// SIMATIC STEP 7 (V5.x) project 2800
// CPU: CPU 315-2 DP
// station: P_ADR_BUS
// station: Hardware
// station: SIMATIC 300(1)
// program: S7 Program(1)

SYMBOL_TABLE
"CLOCK_OP"	DB 5	DB 5	// COMMUNICATION CLOCK OP
"TransferValves"	DB 10	DB 10	// Data Transfer for Valves
"TransferMotor"	DB 11	DB 11	// Data Transfer for Motor
"TransferLevel"	DB 12	DB 12	// Data Transfer for Level
"TransferTemperature"	DB 14	DB 14	// Data Transfer for Temperatuer
"TransferPID"	DB 15	DB 15	// Data Transfer for PID
"TransferFlow"	DB 16	DB 16	// Data Transfer for Flow
"TransferWeight"	DB 18	DB 18	// Data Transfer for Weight
"TransferGenerell"	DB 30	DB 30	// Data Transfer Generell
"TransferRecipe"	DB 90	DB 90	// Data Transfer for Recipe
"TransferBatch"	DB 91	DB 91	// Data Transfer for Batch
"DataBatchControl"	DB 92	FB 90
"ALARMTIME"	DB 100	DB 100	// actual timers alarms
"ALARMBLOCK"	DB 110	DB 110	// alarm indication to OP
"ALARM_ACK_OP"	DB 115	DB 115	// alarm acknowledge from OP
"LAMPS_ACK"	DB 120	DB 120	// lamp acknowledge
"CLOCK_FB"	FB 5	FB 5	// SETTING CPU CLOCK
"preparation"	FB 10	FB 10	// starch preparation
"Devices"	FB 20	FB 20	// Devices
"ALARM_HANDLING"	FB 31	FB 31	// alarm handling
"ALARM"	FB 33	FB 33	// indication alarm
"Batch"	FB 90	FB 90	// Batch
"BatchControl"	FC 10	FC 10	// Batch Control
"RecipeControl"	FC 90	FC 90	// Recipe Control
"DosLine"	FC 91	FC 91	// Dosing Line
"AUTO_VALVE"	FC 100	FC 100	// automatic valve
"MOTOR"	FC 101	FC 101	// motor control
"level"	FC 107	FC 107	// level display
"temperature"	FC 109	FC 109	// temperature display
"AI_4-20"	FC 111	FC 111	// analog input 4-20mA
"weight"	FC 114	FC 114	// weighing unit
"ALARM_BLOCK"	FC 115	FC 115	// alarm function block
"M22_01_RUN"	I 4.0	BOOL	// screw conveyor sizing starch running
"M23_01_RUN"	I 4.1	BOOL	// dedusting station sizing starch running
"M24_01_RUN"	I 4.2	BOOL	// agitator cooker sizing starch running
"M25_01_RUN"	I 4.3	BOOL	// pump sizing starch running
"M26_01_RUN"	I 4.4	BOOL	// stby pump sizing starch running
"HS22_02_ZSC"	I 4.5	BOOL	// valve screw conveyor sizing starch closed
"HS22_02_ZSO"	I 4.6	BOOL	// valve screw conveyor sizing starch open
"HS24_06_ZSC"	I 4.7	BOOL	// water valve cooker sizing starch closed
"HS24_08_ZSC"	I 5.0	BOOL	// discharge valve cooker sizing starch closed
"XS28_02_K1"	I 5.1	BOOL	// release filling storage tank sizing starch
"Signal_0"	M 1.0	BOOL	// Signal 0
"Signal_1"	M 1.1	BOOL	// Signal 1
"1_second"	M 1.2	BOOL	// second pulse
"PB_LAMP_ACK"	M 1.3	BOOL	// Lamp acknowledge
"spike_ pulse_ 1H"	M 2.0	BOOL	// spike pulse 1 houre
"Release_Time"	M 2.1	BOOL	// release timetransfer
"Pulse_Time"	M 2.2	BOOL	// pulse timetransfer
"OP_COMM_OK"	M 9.0	BOOL	// Op Communication ok
"LB_OP_PULS"	M 9.1	BOOL
"fault_M_22_01"	M 12.0	BOOL	// fault motor M 22.01
"fault_M_23_01"	M 12.1	BOOL	// fault motor M 23.01
"fault_M_24_01"	M 12.2	BOOL	// fault motor M 24.01
"fault_M_25_01"	M 12.3	BOOL	// fault motor M 25.01
"fault_M_26_01"	M 12.4	BOOL	// fault motor M 26.01
"fault_HS_22_02"	M 14.0	BOOL	// fault valve HS 22.02
"fault_HS_22_06"	M 14.1	BOOL	// fault valve HS 22.06
"fault_HS_24_06"	M 14.2	BOOL	// fault valve HS 24.06
"fault_HS_24_07"	M 14.3	BOOL	// fault valve HS 24.07
"fault_HS_24_08"	M 14.4	BOOL	// fault valve HS 24.08
"fault_WQ_24_04"	M 16.0	BOOL	// fault weighing unit WQ 24.04
"fault_TC_24_05"	M 16.1	BOOL	// fault temperature TC 24.05
"fault_XS_28_02"	M 16.2	BOOL	// fault level XS 28.02
"fault_HH_WQ_24_04"	M 17.0	BOOL	// fault alarm high weighing unit WQ 24.04
"fault_HH_TC_24_05"	M 17.1	BOOL	// fault alarm high temperature TC 24.05
"fault_HH_XS_28_02"	M 17.2	BOOL	// fault alarm high level XS 28.02
"fault_LL_XS_28_02"	M 17.3	BOOL	// fault alarm low level XS 28.02
"HH_WQ_24_04"	M 60.0	BOOL	// Alarm HH WQ 24.04
"HH_TC_24_05"	M 60.1	BOOL	// Alarm HH TC 24.05
"HH_XS_28_02"	M 60.2	BOOL	// Alarm HH XS 28.02
"H_WQ_24_05"	M 61.0	BOOL	// Alarm H WQ 24.05
"H_TC_24_05"	M 61.1	BOOL	// Alarm H TC 24.05
"H_XS_28_02"	M 61.2	BOOL	// Alarm H XS 28.02
"L_WQ_24_06"	M 62.0	BOOL	// Alarm L WQ 24.06
"L_TC_24_05"	M 62.1	BOOL	// Alarm L TC 24.05
"L_XS_28_02"	M 62.2	BOOL	// Alarm L XS 28.02
"LL_WQ_24_07"	M 63.0	BOOL	// Alarm LL WQ 24.07
"LL_TC_24_05"	M 63.1	BOOL	// Alarm LL TC 24.05
"LL_XS_28_02"	M 63.2	BOOL	// Alarm LL XS 28.02
"check_M_22_01"	M 70.0	BOOL	// check motor M 22.01
"check_M_23_01"	M 70.1	BOOL	// check motor M 23.01
"check_M_24_01"	M 70.2	BOOL	// check motor M 24.01
"check_M_25_01"	M 70.3	BOOL	// check motor M 25.01
"check_M_26_01"	M 70.4	BOOL	// check motor M 26.01
"check_HS_22_02"	M 72.0	BOOL	// check valve HS 22.02
"check_HS_22_06"	M 72.1	BOOL	// check valve HS 22.06
"check_HS_24_06"	M 72.2	BOOL	// check valve HS 24.06
"check_HS_24_07"	M 72.3	BOOL	// check valve HS 24.07
"check_HS_24_08"	M 72.4	BOOL	// check valve HS 24.08
"check_WQ_24_04"	M 74.0	BOOL	// check weight WQ 24.04
"check_TC_24_05"	M 74.1	BOOL	// check temperature TC 24.05
"check_XS_28_02"	M 74.2	BOOL	// check level XS 28.02
"fault_ack_M_22_01"	M 90.0	BOOL	// fault acknowledge motor M 22.01
"fault_ack_M_23_01"	M 90.1	BOOL	// fault acknowledge motor M 23.01
"fault_ack_M_24_01"	M 90.2	BOOL	// fault acknowledge motor M 24.01
"fault_ack_M_25_01"	M 90.3	BOOL	// fault acknowledge motor M 25.01
"fault_ack_M_26_01"	M 90.4	BOOL	// fault acknowledge motor M 26.01
"fault_ack_HS_22_02"	M 92.0	BOOL	// fault acknowledge valve HS 22.02
"fault_ack_HS_22_06"	M 92.1	BOOL	// fault acknowledge valve HS 22.06
"fault_ack_HS_24_06"	M 92.2	BOOL	// fault acknowledge valve HS 24.06
"fault_ack_HS_24_07"	M 92.3	BOOL	// fault acknowledge valve HS 24.07
"fault_ack_HS_24_08"	M 92.4	BOOL	// fault acknowledge valve HS 24.08
"fault_ack_WQ_24_04"	M 94.0	BOOL	// fault acknowledge weight WQ 24.04
"fault_ack_TC_24_05"	M 94.1	BOOL	// fault acknowledge temperature TC 24.05
"fault_ack_XS_28_02"	M 94.2	BOOL	// fault acknowledge level XS 28.02
"fault_ack_HH_WQ_24_04"	M 95.0	BOOL	// fault acknowledge alarm high weighing unit WQ 24.04
"fault_ack_HH_TC_24_05"	M 95.1	BOOL	// fault acknowledge alarm high temperature TC 24.05
"fault_ack_HH_XS_28_02"	M 95.2	BOOL	// fault acknowledge alarm high level XS 28.02
"fault_ack_LL_XS_28_02"	M 95.3	BOOL	// fault acknowledge alarm low level XS 28.02
"auto_on_M_22_01"	M 100.0	BOOL	// auto on motor M 22.01
"auto_on_M_23_01"	M 100.1	BOOL	// auto on motor M 23.01
"auto_on_M_24_01"	M 100.2	BOOL	// auto on motor M 24.01
"auto_on_M_25_01"	M 100.3	BOOL	// auto on motor M 25.01
"auto_on_M_26_01"	M 100.4	BOOL	// auto on motor M 26.01
"auto_on_HS_22_02"	M 102.0	BOOL	// auto on valve HS 22.02
"auto_on_HS_22_06"	M 102.1	BOOL	// auto on valve HS 22.06
"auto_on_HS_24_06"	M 102.2	BOOL	// auto on valve HS 24.06
"auto_on_HS_24_07"	M 102.3	BOOL	// auto on valve HS 24.07
"auto_on_HS_24_08"	M 102.4	BOOL	// auto on valve HS 24.08
"SteamOnEnzym"	M 102.5	BOOL	// Cond. Steam on if Enzymatic Starch selected
"AlarmOnEnzym"	M 102.6	BOOL	// Alarm On Enzym Dosing
"SteamOnHold"	M 102.7	BOOL	// Cond. Steam on at end Temperaturcontrol
"LockSelModified"	M 110.0	BOOL	// Lock Selection Button if Batch is running
"Cond_Dos_Starch"	M 120.0	BOOL	// Condition Dosing Starch
"Save_Dil_On_Starch"	M 120.1	BOOL	// Save Dilution was on starch
"Agitator_Stop_Starch"	M 120.2	BOOL	// Agitator stop starch
"Save_Dis_On_Starch"	M 120.3	BOOL	// Save discharge was on starch
"IMP_START_STARCH"	M 160.0	BOOL	// Impuls Start Batch Starch
"Hold_Mixing_Time_Starch"	M 160.1	BOOL	// Hold Mixing Time Starch
"Discharged1_Starch"	M 161.0	BOOL	// Discharged 1 starch
"Discharged2_Starch"	M 161.1	BOOL	// Discharged 2 starch
"Batch_Starch_Running"	M 180.0	BOOL	// Batch Starch Running
"Batch_Starch_Started"	M 180.1	BOOL	// Batch Starch Started
"Dos_On_Water_Starch"	M 185.0	BOOL	// Dosing on water starch
"Cmd_Agitator_On_Starch"	M 185.1	BOOL	// Command Agitator on starch
"Dos_On_Powder_Starch"	M 185.2	BOOL	// Dosing on powder starch
"Dos_On_Steam_Starch"	M 185.3	BOOL	// Dosing on steam starch
"Dos_On_Dil_Water_Starch"	M 185.4	BOOL	// Dosing on dilution water starch
"Cmd_Discharge1_On_Starch"	M 185.5	BOOL	// Command discharge 1 on starch
"Active_Discharge1_Starch"	M 185.6	BOOL	// Active Discharge 1 Starch
"Dos_On_Flushwater_Starch"	M 185.7	BOOL	// Dosing on flushwater starch
"Cmd_Discharge2_On_Starch"	M 186.0	BOOL	// Command discharge 2 on starch
"Active_Discharge2_Starch"	M 186.1	BOOL	// Active Discharge 2 Starch
"Active_Dil_Water_Starch"	M 186.2	BOOL	// Dosing active dilution water starch
"Cmd_Enzym_On_Starch"	M 186.3	BOOL	// Dosing Enzym Request
"Enzyme_Done_Starch"	M 186.4	BOOL	// Enzym finished
"Dos_On_EnzSteam_Starch"	M 186.5	BOOL	// Dosing on Steam for Enzymatic Starch
"Active_Hold_Temp_Starch"	M 186.6	BOOL	// Holding Temperature active Enzymatic Starch
"Active_Temp_Starch"	M 186.7	BOOL	// Temperature Hold at end of Starch
"WQ_24_04_Value"	MD 30	REAL	// value WQ 24.04
"TC_24_05_Value"	MD 34	REAL	// value TC 24.05
"XS_28_02_Value"	MD 38	REAL	// value percent XS 28.02
"Cycle_Time"	MW 252	INT	// Cycle Time
"WQ24_04_IN"	PIW 256	WORD	// weight cooker sizing starch
"XS28_02_LI"	PIW 258	WORD	// level storage tank cooked sizing starch
"TC24_05_IN"	PIW 260	WORD	// temperature cooker sizing starch
"M22_01_ON"	Q 8.0	BOOL	// screw conveyor sizing starch on
"M23_01_ON"	Q 8.1	BOOL	// dedusting station sizing starch on
"M23_01_ST"	Q 8.2	BOOL	// dedusting station sizing starch on
"M24_01_ON"	Q 8.3	BOOL	// agitator cooker sizing starch on
"M25_01_ON"	Q 8.4	BOOL	// pump sizing starch on
"M26_01_ON"	Q 8.5	BOOL	// stby pump sizing starch on
"HS22_02_ON"	Q 8.6	BOOL	// valve screw conveyor sizing starch on
"HS22_06_ON"	Q 8.7	BOOL	// air valve screw conveyor sizing starch on
"HS24_06_ON"	Q 9.0	BOOL	// water valve cooker sizing starch on
"HS24_07_ON"	Q 9.1	BOOL	// steam valve cooker sizing starch on
"HS24_08_ON"	Q 9.2	BOOL	// discharge valve cooker sizing starch on
"XA28_01_ON"	Q 9.3	BOOL	// alarm preparation on
"XS28_02_K2"	Q 9.4	BOOL	// filling is on storage tank sizing starch
"XS28_02_K3"	Q 9.5	BOOL	// fault filling storage tank sizing starch
"SET_CLK"	SFC 0	SFC 0	// Set System Clock
"Valve UDT"	UDT 1	UDT 1	// Data Valve
"Valve Popup UDT"	UDT 2	UDT 2	// Data Valve Popup
"Motor UDT"	UDT 3	UDT 3	// Data Motor
"Motor Popup UDT"	UDT 4	UDT 4	// Data Motor Popup
"Level UDT"	UDT 5	UDT 5	// Data Level
"Level Popup UDT"	UDT 6	UDT 6	// Data Level Popup
"Pressure UDT"	UDT 7	UDT 7	// Data Pressure
"Pressure Popup UDT"	UDT 8	UDT 8	// Data Pressure Popup
"Temperature UDT"	UDT 9	UDT 9	// Data Temperature
"Temperature Popup UDT"	UDT 10	UDT 10	// Data Temperature Popup
"Controler UDT"	UDT 11	UDT 11	// Data Controler
"Controler Popup UDT"	UDT 12	UDT 12	// Data Controler Popup
"Flow UDT"	UDT 13	UDT 13	// Data Flow
"Flow Popup UDT"	UDT 14	UDT 14	// Data Flow Popup
"Viskosity UDT"	UDT 15	UDT 15	// Viskosity Data
"Viskosity Popup UDT"	UDT 16	UDT 16	// Data Viskosity Popup
"Weight UDT"	UDT 17	UDT 17	// Weight Data
"Weight Popup UDT"	UDT 18	UDT 18	// Data Weight Popup
"Recipe UDT"	UDT 90	UDT 90	// Data Recipe
"DosLine UDT"	UDT 91	UDT 91	// Dosing Line UDT
END_SYMBOL_TABLE

FUNCTION_BLOCK "CLOCK_FB"	// FB 5
AUTHOR : gaw-be
FAMILY : GAW
NAME : DATETIME
VERSION : 0.1
BEGIN
// (block stored without names or comments; labels and parameter names are numbered)
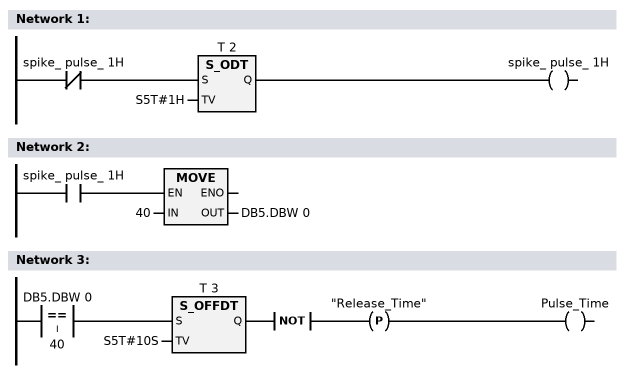
NETWORK
TITLE =
      AN    "spike_ pulse_ 1H";
      L     S5T#1H;
      SD    T 2;
      NOP   0;
      NOP   0;
      NOP   0;
      A     T 2;
      =     "spike_ pulse_ 1H";
NETWORK
TITLE =
      A     "spike_ pulse_ 1H";
      JNB   M001;
      L     40;
      T     DB5.DBW 0;
M001: NOP   0;
NETWORK
TITLE =
      A(;
      A(;
      L     DB5.DBW 0;
      L     40;
      ==I;
      );
      L     S5T#10S;
      SF    T 3;
      NOP   0;
      NOP   0;
      NOP   0;
      A     T 3;
      );
      NOT;
      FP    "Release_Time";
      =     "Pulse_Time";
NETWORK
TITLE =
      A     "Pulse_Time";
      JNB   M002;
      BLD   7;
      L     5;
      T     LW 102;
      L     P#DBX 8.0;
      T     LD 104;
      UC    "SET_CLK";
      {     P#L 102.0, P#L 100.0 };
      BLD   8;
M002: NOP   0;
END_FUNCTION_BLOCK

FUNCTION_BLOCK "preparation"	// FB 10
VERSION : 0.1
BEGIN
// (block stored without names or comments; labels and parameter names are numbered)
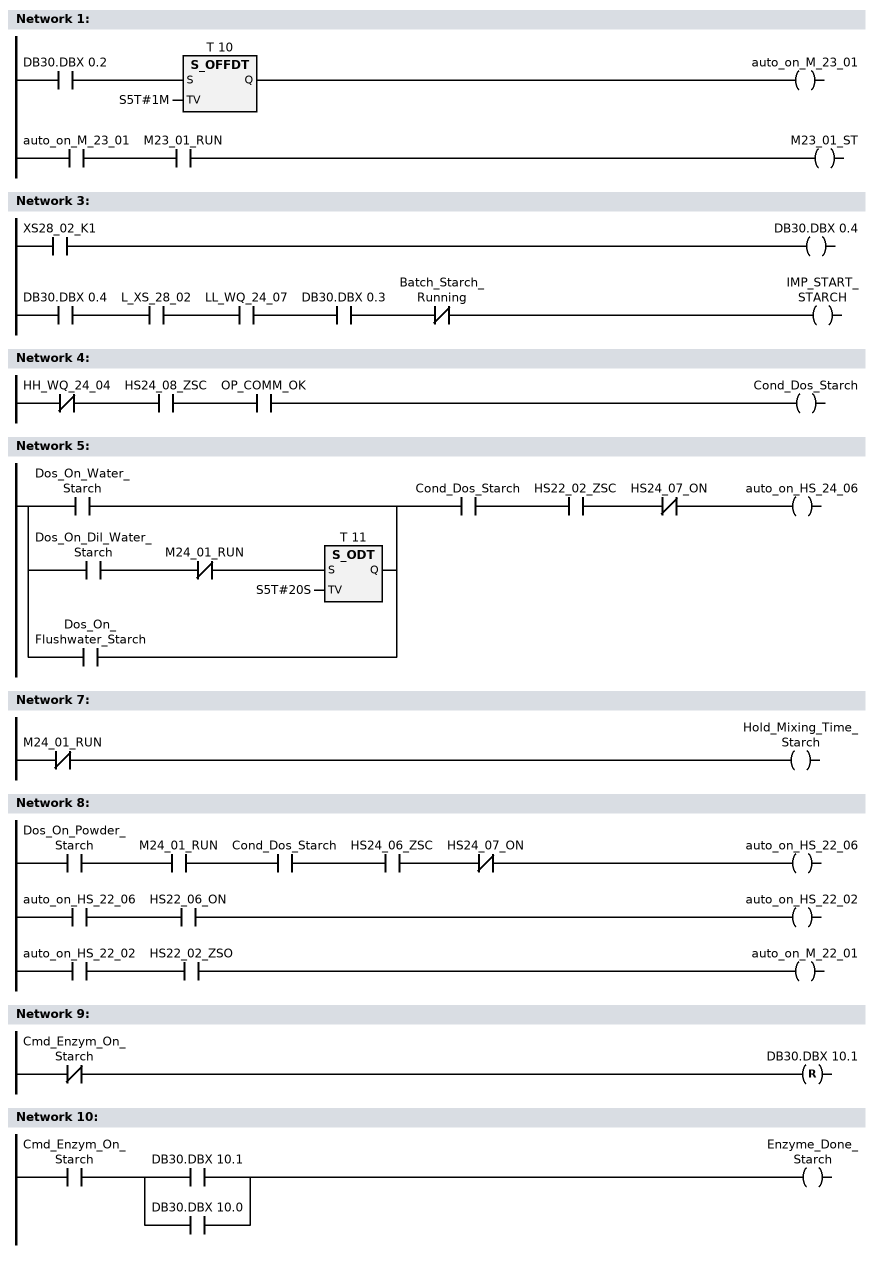
NETWORK
TITLE =
      A(;
      A     DB30.DBX 0.2;
      L     S5T#1M;
      SF    T 10;
      NOP   0;
      NOP   0;
      NOP   0;
      A     T 10;
      );
      =     "auto_on_M_23_01";
      A     "auto_on_M_23_01";
      A     "M23_01_RUN";
      =     "M23_01_ST";
NETWORK
TITLE =
      AN    "Batch_Starch_Running";
      A     DB30.DBX 10.0;
      S     "LockSelModified";
      AN    "Batch_Starch_Running";
      AN    DB30.DBX 10.0;
      R     "LockSelModified";
      A     "LockSelModified";
      =     L 8.0;
      A     L 8.0;
      A     "Batch_Starch_Running";
      S     DB30.DBX 10.0;
      AN    L 8.0;
      A     "Batch_Starch_Running";
      R     DB30.DBX 10.0;
NETWORK
TITLE =
      A     "XS28_02_K1";
      =     DB30.DBX 0.4;
      A     DB30.DBX 0.4;
      A     "L_XS_28_02";
      A     "LL_WQ_24_07";
      A     DB30.DBX 0.3;
      AN    "Batch_Starch_Running";
      =     "IMP_START_STARCH";
NETWORK
TITLE =
      AN    "HH_WQ_24_04";
      A     "HS24_08_ZSC";
      A     "OP_COMM_OK";
      =     "Cond_Dos_Starch";
NETWORK
TITLE =
      A(;
      O     "Dos_On_Water_Starch";
      O(;
      A     "Dos_On_Dil_Water_Starch";
      AN    "M24_01_RUN";
      L     S5T#20S;
      SD    T 11;
      NOP   0;
      NOP   0;
      NOP   0;
      A     T 11;
      );
      O     "Dos_On_Flushwater_Starch";
      );
      A     "Cond_Dos_Starch";
      A     "HS22_02_ZSC";
      AN    "HS24_07_ON";
      =     "auto_on_HS_24_06";
NETWORK
TITLE =
      AN    "LL_WQ_24_07";
      A     "Cmd_Agitator_On_Starch";
      A(;
      A(;
      A     "Dos_On_Dil_Water_Starch";
      S     "Save_Dil_On_Starch";
      AN    "Active_Dil_Water_Starch";
      R     "Save_Dil_On_Starch";
      A     "Save_Dil_On_Starch";
      );
      NOT;
      );
      A(;
      A(;
      A     "Cmd_Discharge1_On_Starch";
      A     "L_WQ_24_06";
      S     "Agitator_Stop_Starch";
      AN    "Batch_Starch_Running";
      R     "Agitator_Stop_Starch";
      A     "Agitator_Stop_Starch";
      );
      NOT;
      );
      =     "auto_on_M_24_01";
NETWORK
TITLE =
      AN    "M24_01_RUN";
      =     "Hold_Mixing_Time_Starch";
NETWORK
TITLE =
      A     "Dos_On_Powder_Starch";
      A     "M24_01_RUN";
      A     "Cond_Dos_Starch";
      A     "HS24_06_ZSC";
      AN    "HS24_07_ON";
      =     "auto_on_HS_22_06";
      A     "auto_on_HS_22_06";
      A     "HS22_06_ON";
      =     "auto_on_HS_22_02";
      A     "auto_on_HS_22_02";
      A     "HS22_02_ZSO";
      =     "auto_on_M_22_01";
NETWORK
TITLE =
      AN    "Cmd_Enzym_On_Starch";
      R     DB30.DBX 10.1;
NETWORK
TITLE =
      A     "Cmd_Enzym_On_Starch";
      A(;
      O     DB30.DBX 10.1;
      O     DB30.DBX 10.0;
      );
      =     "Enzyme_Done_Starch";
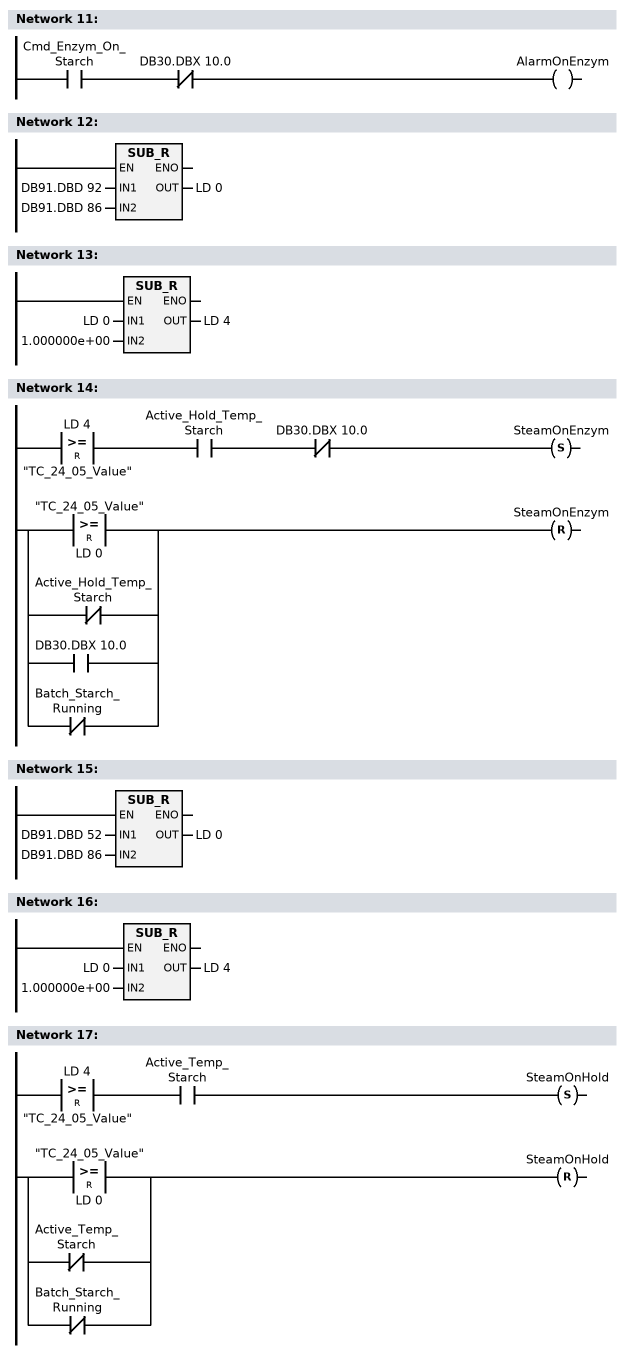
NETWORK
TITLE =
      A     "Cmd_Enzym_On_Starch";
      AN    DB30.DBX 10.0;
      =     "AlarmOnEnzym";
NETWORK
TITLE =
      L     DB91.DBD 92;
      L     DB91.DBD 86;
      -R;
      T     LD 0;
      NOP   0;
NETWORK
TITLE =
      L     LD 0;
      L     1.000000e+00;
      -R;
      T     LD 4;
      NOP   0;
NETWORK
TITLE =
      A(;
      L     LD 4;
      L     "TC_24_05_Value";
      >=R;
      );
      A     "Active_Hold_Temp_Starch";
      AN    DB30.DBX 10.0;
      S     "SteamOnEnzym";
      A(;
      O(;
      L     "TC_24_05_Value";
      L     LD 0;
      >=R;
      );
      ON    "Active_Hold_Temp_Starch";
      O     DB30.DBX 10.0;
      ON    "Batch_Starch_Running";
      );
      R     "SteamOnEnzym";
      NOP   0;
NETWORK
TITLE =
      L     DB91.DBD 52;
      L     DB91.DBD 86;
      -R;
      T     LD 0;
      NOP   0;
NETWORK
TITLE =
      L     LD 0;
      L     1.000000e+00;
      -R;
      T     LD 4;
      NOP   0;
NETWORK
TITLE =
      A(;
      L     LD 4;
      L     "TC_24_05_Value";
      >=R;
      );
      A     "Active_Temp_Starch";
      S     "SteamOnHold";
      A(;
      O(;
      L     "TC_24_05_Value";
      L     LD 0;
      >=R;
      );
      ON    "Active_Temp_Starch";
      ON    "Batch_Starch_Running";
      );
      R     "SteamOnHold";
      NOP   0;
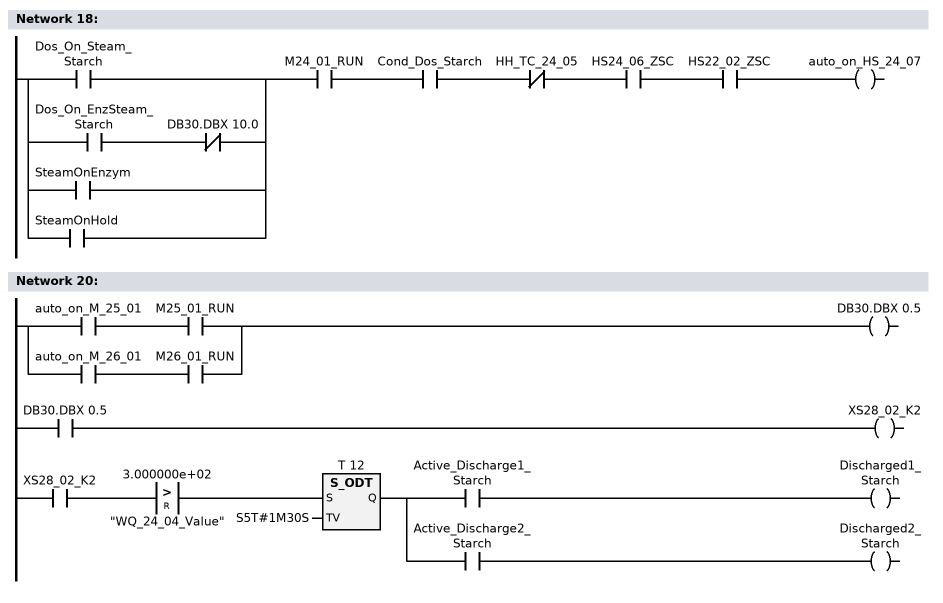
NETWORK
TITLE =
      A(;
      O     "Dos_On_Steam_Starch";
      O;
      A     "Dos_On_EnzSteam_Starch";
      AN    DB30.DBX 10.0;
      O     "SteamOnEnzym";
      O     "SteamOnHold";
      );
      A     "M24_01_RUN";
      A     "Cond_Dos_Starch";
      AN    "HH_TC_24_05";
      A     "HS24_06_ZSC";
      A     "HS22_02_ZSC";
      =     "auto_on_HS_24_07";
NETWORK
TITLE =
      A(;
      A(;
      A     "XS28_02_K1";
      A     "L_XS_28_02";
      O(;
      A     "auto_on_HS_24_08";
      A     "Active_Discharge1_Starch";
      S     "Save_Dis_On_Starch";
      AN    "Active_Discharge1_Starch";
      R     "Save_Dis_On_Starch";
      A     "Save_Dis_On_Starch";
      );
      );
      A     "Cmd_Discharge1_On_Starch";
      A     "Active_Discharge1_Starch";
      O;
      A     "Cmd_Discharge2_On_Starch";
      A     "Active_Discharge2_Starch";
      );
      AN    "HH_XS_28_02";
      =     "auto_on_HS_24_08";
      A     "auto_on_HS_24_08";
      AN    "HS24_08_ZSC";
      =     L 8.0;
      A     L 8.0;
      AN    DB30.DBX 0.0;
      =     "auto_on_M_25_01";
      A     L 8.0;
      A     DB30.DBX 0.0;
      =     "auto_on_M_26_01";
NETWORK
TITLE =
      A(;
      A     "auto_on_M_25_01";
      A     "M25_01_RUN";
      O;
      A     "auto_on_M_26_01";
      A     "M26_01_RUN";
      );
      =     DB30.DBX 0.5;
      A     DB30.DBX 0.5;
      =     "XS28_02_K2";
      A     "XS28_02_K2";
      A(;
      L     3.000000e+02;
      L     "WQ_24_04_Value";
      >R;
      );
      L     S5T#1M30S;
      SD    T 12;
      NOP   0;
      NOP   0;
      NOP   0;
      A     T 12;
      =     L 8.0;
      A     L 8.0;
      A     "Active_Discharge1_Starch";
      =     "Discharged1_Starch";
      A     L 8.0;
      A     "Active_Discharge2_Starch";
      =     "Discharged2_Starch";
END_FUNCTION_BLOCK

FUNCTION_BLOCK "Devices"	// FB 20
VERSION : 0.1
BEGIN
// (block stored without names or comments; labels and parameter names are numbered)
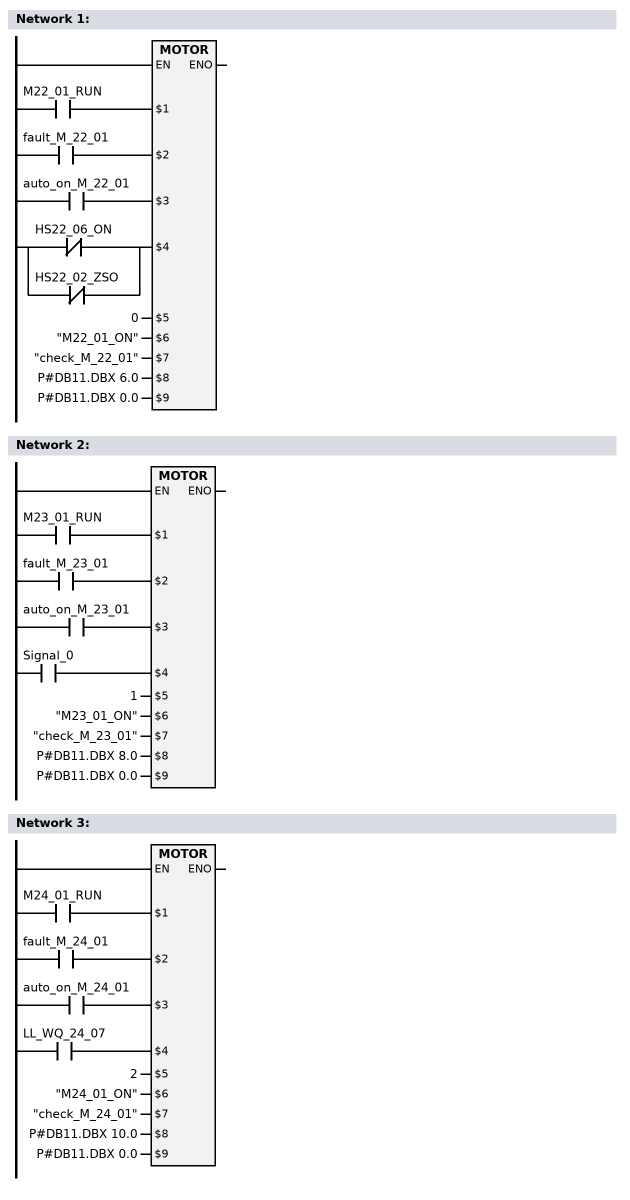
NETWORK
TITLE =
      A     "M22_01_RUN";
      =     L 18.0;
      BLD   103;
      A     "fault_M_22_01";
      =     L 18.1;
      BLD   103;
      A     "auto_on_M_22_01";
      =     L 18.2;
      BLD   103;
      A(;
      ON    "HS22_06_ON";
      ON    "HS22_02_ZSO";
      );
      =     L 18.3;
      BLD   103;
      CALL  "MOTOR" (
           $1                       := L 18.0,
           $2                       := L 18.1,
           $3                       := L 18.2,
           $4                       := L 18.3,
           $5                       := 0,
           $6                       := "M22_01_ON",
           $7                       := "check_M_22_01",
           $8                       := P#DB11.DBX 6.0,
           $9                       := P#DB11.DBX 0.0);
      NOP   0;
NETWORK
TITLE =
      A     "M23_01_RUN";
      =     L 18.0;
      BLD   103;
      A     "fault_M_23_01";
      =     L 18.1;
      BLD   103;
      A     "auto_on_M_23_01";
      =     L 18.2;
      BLD   103;
      A     "Signal_0";
      =     L 18.3;
      BLD   103;
      CALL  "MOTOR" (
           $1                       := L 18.0,
           $2                       := L 18.1,
           $3                       := L 18.2,
           $4                       := L 18.3,
           $5                       := 1,
           $6                       := "M23_01_ON",
           $7                       := "check_M_23_01",
           $8                       := P#DB11.DBX 8.0,
           $9                       := P#DB11.DBX 0.0);
      NOP   0;
NETWORK
TITLE =
      A     "M24_01_RUN";
      =     L 18.0;
      BLD   103;
      A     "fault_M_24_01";
      =     L 18.1;
      BLD   103;
      A     "auto_on_M_24_01";
      =     L 18.2;
      BLD   103;
      A     "LL_WQ_24_07";
      =     L 18.3;
      BLD   103;
      CALL  "MOTOR" (
           $1                       := L 18.0,
           $2                       := L 18.1,
           $3                       := L 18.2,
           $4                       := L 18.3,
           $5                       := 2,
           $6                       := "M24_01_ON",
           $7                       := "check_M_24_01",
           $8                       := P#DB11.DBX 10.0,
           $9                       := P#DB11.DBX 0.0);
      NOP   0;
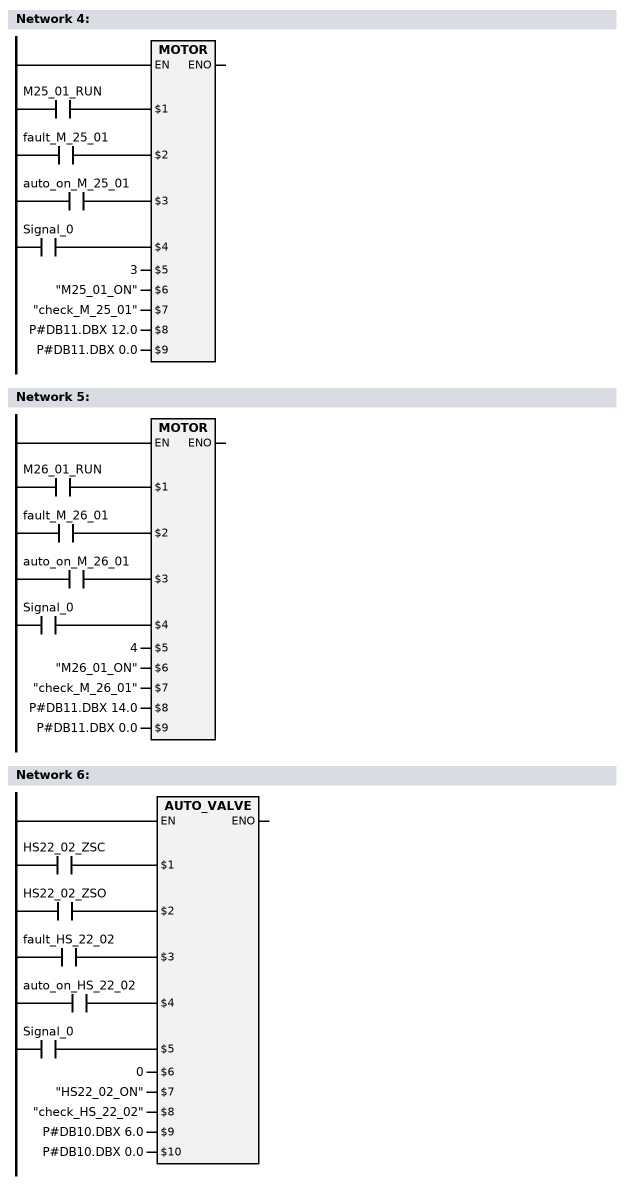
NETWORK
TITLE =
      A     "M25_01_RUN";
      =     L 18.0;
      BLD   103;
      A     "fault_M_25_01";
      =     L 18.1;
      BLD   103;
      A     "auto_on_M_25_01";
      =     L 18.2;
      BLD   103;
      A     "Signal_0";
      =     L 18.3;
      BLD   103;
      CALL  "MOTOR" (
           $1                       := L 18.0,
           $2                       := L 18.1,
           $3                       := L 18.2,
           $4                       := L 18.3,
           $5                       := 3,
           $6                       := "M25_01_ON",
           $7                       := "check_M_25_01",
           $8                       := P#DB11.DBX 12.0,
           $9                       := P#DB11.DBX 0.0);
      NOP   0;
NETWORK
TITLE =
      A     "M26_01_RUN";
      =     L 18.0;
      BLD   103;
      A     "fault_M_26_01";
      =     L 18.1;
      BLD   103;
      A     "auto_on_M_26_01";
      =     L 18.2;
      BLD   103;
      A     "Signal_0";
      =     L 18.3;
      BLD   103;
      CALL  "MOTOR" (
           $1                       := L 18.0,
           $2                       := L 18.1,
           $3                       := L 18.2,
           $4                       := L 18.3,
           $5                       := 4,
           $6                       := "M26_01_ON",
           $7                       := "check_M_26_01",
           $8                       := P#DB11.DBX 14.0,
           $9                       := P#DB11.DBX 0.0);
      NOP   0;
NETWORK
TITLE =
      A     "HS22_02_ZSC";
      =     L 18.0;
      BLD   103;
      A     "HS22_02_ZSO";
      =     L 18.1;
      BLD   103;
      A     "fault_HS_22_02";
      =     L 18.2;
      BLD   103;
      A     "auto_on_HS_22_02";
      =     L 18.3;
      BLD   103;
      A     "Signal_0";
      =     L 18.4;
      BLD   103;
      CALL  "AUTO_VALVE" (
           $1                       := L 18.0,
           $2                       := L 18.1,
           $3                       := L 18.2,
           $4                       := L 18.3,
           $5                       := L 18.4,
           $6                       := 0,
           $7                       := "HS22_02_ON",
           $8                       := "check_HS_22_02",
           $9                       := P#DB10.DBX 6.0,
           $10                      := P#DB10.DBX 0.0);
      NOP   0;
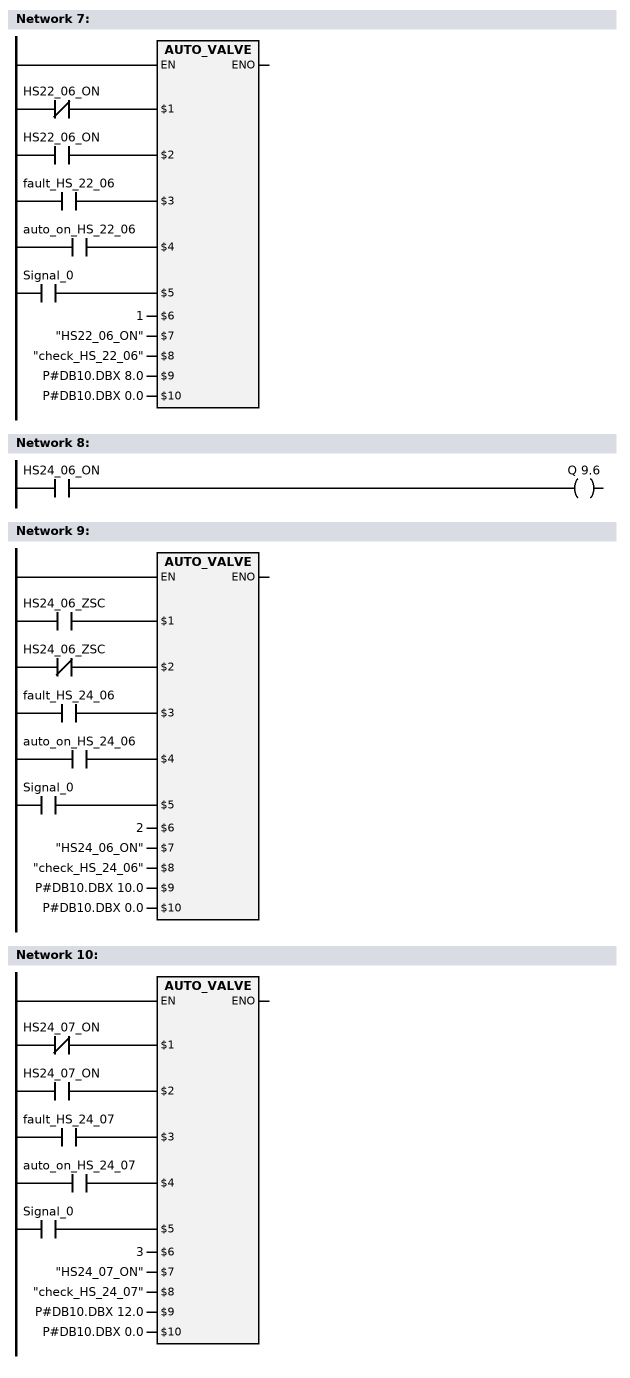
NETWORK
TITLE =
      AN    "HS22_06_ON";
      =     L 18.0;
      BLD   103;
      A     "HS22_06_ON";
      =     L 18.1;
      BLD   103;
      A     "fault_HS_22_06";
      =     L 18.2;
      BLD   103;
      A     "auto_on_HS_22_06";
      =     L 18.3;
      BLD   103;
      A     "Signal_0";
      =     L 18.4;
      BLD   103;
      CALL  "AUTO_VALVE" (
           $1                       := L 18.0,
           $2                       := L 18.1,
           $3                       := L 18.2,
           $4                       := L 18.3,
           $5                       := L 18.4,
           $6                       := 1,
           $7                       := "HS22_06_ON",
           $8                       := "check_HS_22_06",
           $9                       := P#DB10.DBX 8.0,
           $10                      := P#DB10.DBX 0.0);
      NOP   0;
NETWORK
TITLE =
      A     "HS24_06_ON";
      =     Q 9.6;
NETWORK
TITLE =
      A     "HS24_06_ZSC";
      =     L 18.0;
      BLD   103;
      AN    "HS24_06_ZSC";
      =     L 18.1;
      BLD   103;
      A     "fault_HS_24_06";
      =     L 18.2;
      BLD   103;
      A     "auto_on_HS_24_06";
      =     L 18.3;
      BLD   103;
      A     "Signal_0";
      =     L 18.4;
      BLD   103;
      CALL  "AUTO_VALVE" (
           $1                       := L 18.0,
           $2                       := L 18.1,
           $3                       := L 18.2,
           $4                       := L 18.3,
           $5                       := L 18.4,
           $6                       := 2,
           $7                       := "HS24_06_ON",
           $8                       := "check_HS_24_06",
           $9                       := P#DB10.DBX 10.0,
           $10                      := P#DB10.DBX 0.0);
      NOP   0;
NETWORK
TITLE =
      AN    "HS24_07_ON";
      =     L 18.0;
      BLD   103;
      A     "HS24_07_ON";
      =     L 18.1;
      BLD   103;
      A     "fault_HS_24_07";
      =     L 18.2;
      BLD   103;
      A     "auto_on_HS_24_07";
      =     L 18.3;
      BLD   103;
      A     "Signal_0";
      =     L 18.4;
      BLD   103;
      CALL  "AUTO_VALVE" (
           $1                       := L 18.0,
           $2                       := L 18.1,
           $3                       := L 18.2,
           $4                       := L 18.3,
           $5                       := L 18.4,
           $6                       := 3,
           $7                       := "HS24_07_ON",
           $8                       := "check_HS_24_07",
           $9                       := P#DB10.DBX 12.0,
           $10                      := P#DB10.DBX 0.0);
      NOP   0;
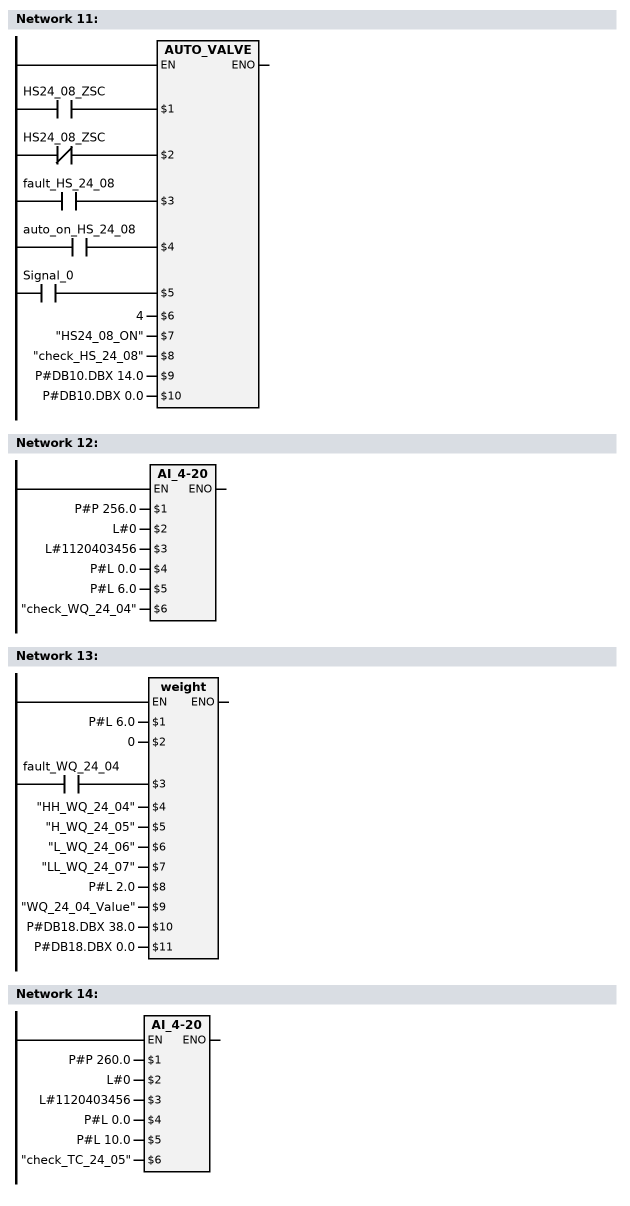
NETWORK
TITLE =
      A     "HS24_08_ZSC";
      =     L 18.0;
      BLD   103;
      AN    "HS24_08_ZSC";
      =     L 18.1;
      BLD   103;
      A     "fault_HS_24_08";
      =     L 18.2;
      BLD   103;
      A     "auto_on_HS_24_08";
      =     L 18.3;
      BLD   103;
      A     "Signal_0";
      =     L 18.4;
      BLD   103;
      CALL  "AUTO_VALVE" (
           $1                       := L 18.0,
           $2                       := L 18.1,
           $3                       := L 18.2,
           $4                       := L 18.3,
           $5                       := L 18.4,
           $6                       := 4,
           $7                       := "HS24_08_ON",
           $8                       := "check_HS_24_08",
           $9                       := P#DB10.DBX 14.0,
           $10                      := P#DB10.DBX 0.0);
      NOP   0;
NETWORK
TITLE =
      CALL  "AI_4-20" (
           $1                       := P#P 256.0,
           $2                       := L#0,
           $3                       := L#1120403456,
           $4                       := P#L 0.0,
           $5                       := P#L 6.0,
           $6                       := "check_WQ_24_04");
      NOP   0;
NETWORK
TITLE =
      A     "fault_WQ_24_04";
      =     L 18.0;
      BLD   103;
      CALL  "weight" (
           $1                       := P#L 6.0,
           $2                       := 0,
           $3                       := L 18.0,
           $4                       := "HH_WQ_24_04",
           $5                       := "H_WQ_24_05",
           $6                       := "L_WQ_24_06",
           $7                       := "LL_WQ_24_07",
           $8                       := P#L 2.0,
           $9                       := "WQ_24_04_Value",
           $10                      := P#DB18.DBX 38.0,
           $11                      := P#DB18.DBX 0.0);
      NOP   0;
NETWORK
TITLE =
      CALL  "AI_4-20" (
           $1                       := P#P 260.0,
           $2                       := L#0,
           $3                       := L#1120403456,
           $4                       := P#L 0.0,
           $5                       := P#L 10.0,
           $6                       := "check_TC_24_05");
      NOP   0;
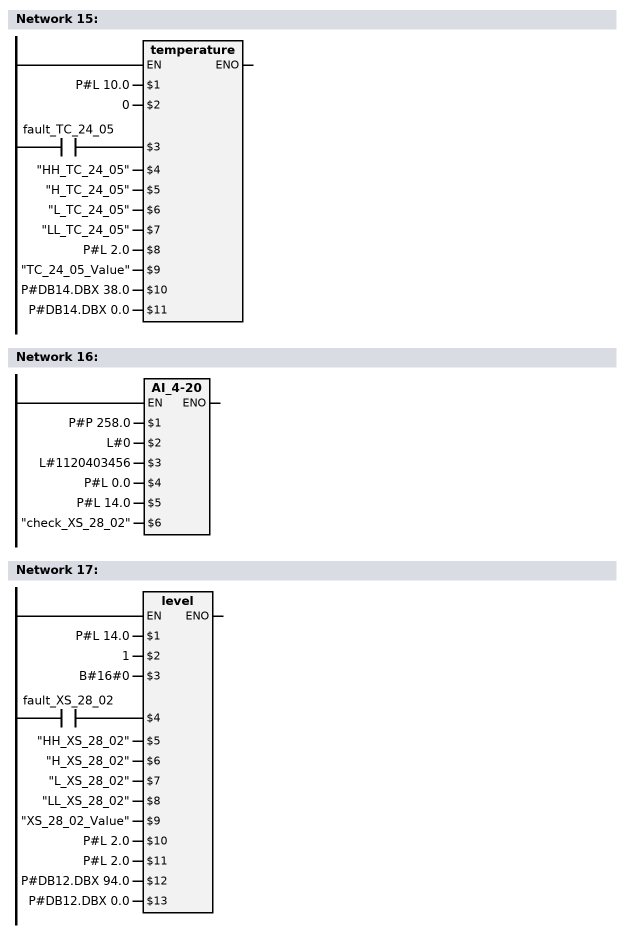
NETWORK
TITLE =
      A     "fault_TC_24_05";
      =     L 18.0;
      BLD   103;
      CALL  "temperature" (
           $1                       := P#L 10.0,
           $2                       := 0,
           $3                       := L 18.0,
           $4                       := "HH_TC_24_05",
           $5                       := "H_TC_24_05",
           $6                       := "L_TC_24_05",
           $7                       := "LL_TC_24_05",
           $8                       := P#L 2.0,
           $9                       := "TC_24_05_Value",
           $10                      := P#DB14.DBX 38.0,
           $11                      := P#DB14.DBX 0.0);
      NOP   0;
NETWORK
TITLE =
      CALL  "AI_4-20" (
           $1                       := P#P 258.0,
           $2                       := L#0,
           $3                       := L#1120403456,
           $4                       := P#L 0.0,
           $5                       := P#L 14.0,
           $6                       := "check_XS_28_02");
      NOP   0;
NETWORK
TITLE =
      A     "fault_XS_28_02";
      =     L 18.0;
      BLD   103;
      CALL  "level" (
           $1                       := P#L 14.0,
           $2                       := 1,
           $3                       := B#16#0,
           $4                       := L 18.0,
           $5                       := "HH_XS_28_02",
           $6                       := "H_XS_28_02",
           $7                       := "L_XS_28_02",
           $8                       := "LL_XS_28_02",
           $9                       := "XS_28_02_Value",
           $10                      := P#L 2.0,
           $11                      := P#L 2.0,
           $12                      := P#DB12.DBX 94.0,
           $13                      := P#DB12.DBX 0.0);
      NOP   0;
END_FUNCTION_BLOCK

FUNCTION_BLOCK "ALARM_HANDLING"	// FB 31
AUTHOR : GAW-LK
FAMILY : ALARM
NAME : ALARMS
VERSION : 0.1
BEGIN
// (block stored without names or comments; labels and parameter names are numbered)
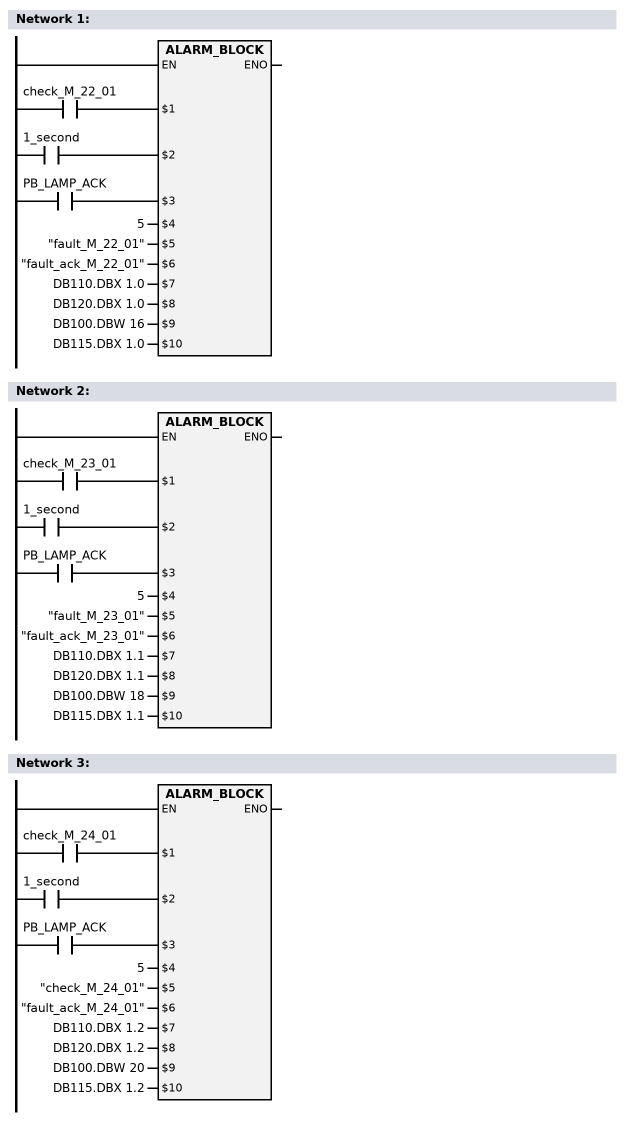
NETWORK
TITLE =
      A     "check_M_22_01";
      =     L 0.0;
      BLD   103;
      A     "1_second";
      =     L 0.1;
      BLD   103;
      A     "PB_LAMP_ACK";
      =     L 0.2;
      BLD   103;
      CALL  "ALARM_BLOCK" (
           $1                       := L 0.0,
           $2                       := L 0.1,
           $3                       := L 0.2,
           $4                       := 5,
           $5                       := "fault_M_22_01",
           $6                       := "fault_ack_M_22_01",
           $7                       := DB110.DBX 1.0,
           $8                       := DB120.DBX 1.0,
           $9                       := DB100.DBW 16,
           $10                      := DB115.DBX 1.0);
      NOP   0;
NETWORK
TITLE =
      A     "check_M_23_01";
      =     L 0.0;
      BLD   103;
      A     "1_second";
      =     L 0.1;
      BLD   103;
      A     "PB_LAMP_ACK";
      =     L 0.2;
      BLD   103;
      CALL  "ALARM_BLOCK" (
           $1                       := L 0.0,
           $2                       := L 0.1,
           $3                       := L 0.2,
           $4                       := 5,
           $5                       := "fault_M_23_01",
           $6                       := "fault_ack_M_23_01",
           $7                       := DB110.DBX 1.1,
           $8                       := DB120.DBX 1.1,
           $9                       := DB100.DBW 18,
           $10                      := DB115.DBX 1.1);
      NOP   0;
NETWORK
TITLE =
      A     "check_M_24_01";
      =     L 0.0;
      BLD   103;
      A     "1_second";
      =     L 0.1;
      BLD   103;
      A     "PB_LAMP_ACK";
      =     L 0.2;
      BLD   103;
      CALL  "ALARM_BLOCK" (
           $1                       := L 0.0,
           $2                       := L 0.1,
           $3                       := L 0.2,
           $4                       := 5,
           $5                       := "check_M_24_01",
           $6                       := "fault_ack_M_24_01",
           $7                       := DB110.DBX 1.2,
           $8                       := DB120.DBX 1.2,
           $9                       := DB100.DBW 20,
           $10                      := DB115.DBX 1.2);
      NOP   0;
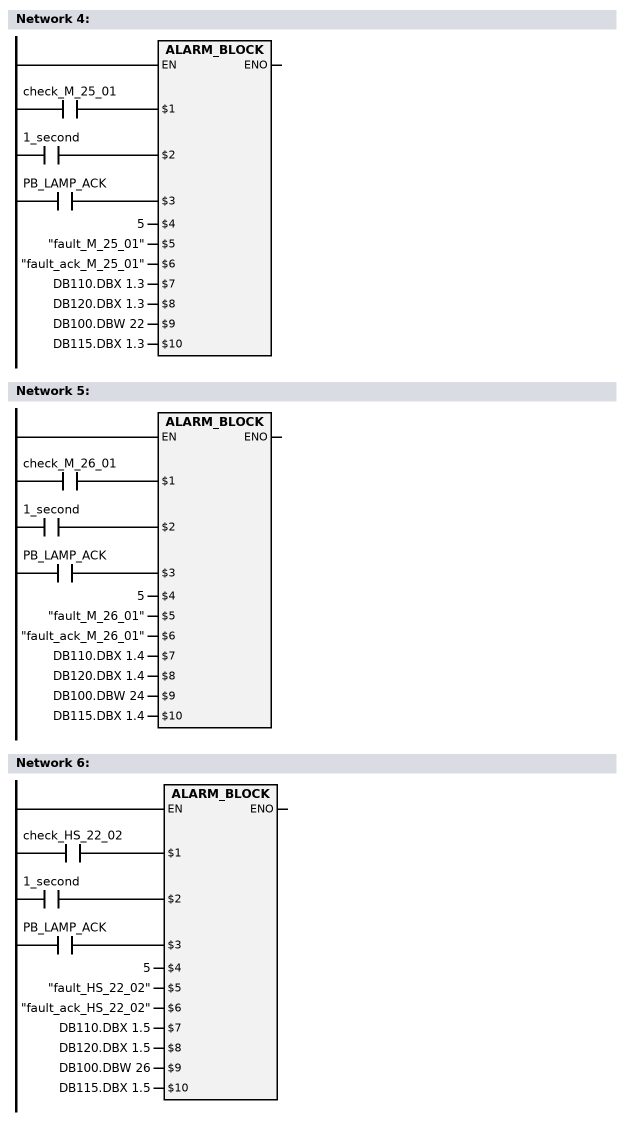
NETWORK
TITLE =
      A     "check_M_25_01";
      =     L 0.0;
      BLD   103;
      A     "1_second";
      =     L 0.1;
      BLD   103;
      A     "PB_LAMP_ACK";
      =     L 0.2;
      BLD   103;
      CALL  "ALARM_BLOCK" (
           $1                       := L 0.0,
           $2                       := L 0.1,
           $3                       := L 0.2,
           $4                       := 5,
           $5                       := "fault_M_25_01",
           $6                       := "fault_ack_M_25_01",
           $7                       := DB110.DBX 1.3,
           $8                       := DB120.DBX 1.3,
           $9                       := DB100.DBW 22,
           $10                      := DB115.DBX 1.3);
      NOP   0;
NETWORK
TITLE =
      A     "check_M_26_01";
      =     L 0.0;
      BLD   103;
      A     "1_second";
      =     L 0.1;
      BLD   103;
      A     "PB_LAMP_ACK";
      =     L 0.2;
      BLD   103;
      CALL  "ALARM_BLOCK" (
           $1                       := L 0.0,
           $2                       := L 0.1,
           $3                       := L 0.2,
           $4                       := 5,
           $5                       := "fault_M_26_01",
           $6                       := "fault_ack_M_26_01",
           $7                       := DB110.DBX 1.4,
           $8                       := DB120.DBX 1.4,
           $9                       := DB100.DBW 24,
           $10                      := DB115.DBX 1.4);
      NOP   0;
NETWORK
TITLE =
      A     "check_HS_22_02";
      =     L 0.0;
      BLD   103;
      A     "1_second";
      =     L 0.1;
      BLD   103;
      A     "PB_LAMP_ACK";
      =     L 0.2;
      BLD   103;
      CALL  "ALARM_BLOCK" (
           $1                       := L 0.0,
           $2                       := L 0.1,
           $3                       := L 0.2,
           $4                       := 5,
           $5                       := "fault_HS_22_02",
           $6                       := "fault_ack_HS_22_02",
           $7                       := DB110.DBX 1.5,
           $8                       := DB120.DBX 1.5,
           $9                       := DB100.DBW 26,
           $10                      := DB115.DBX 1.5);
      NOP   0;
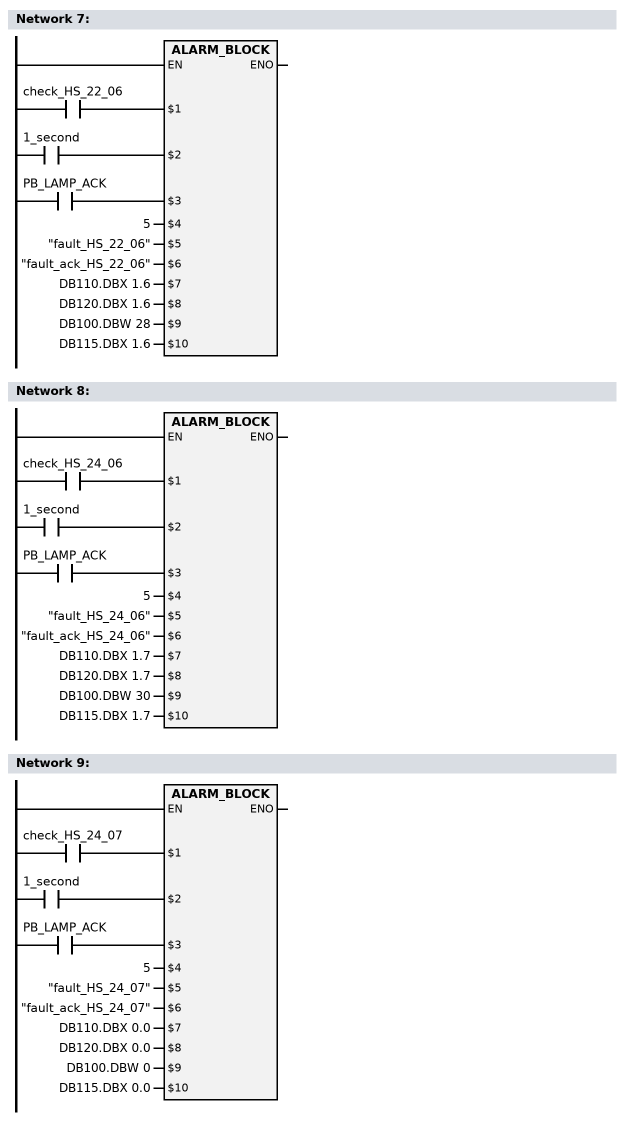
NETWORK
TITLE =
      A     "check_HS_22_06";
      =     L 0.0;
      BLD   103;
      A     "1_second";
      =     L 0.1;
      BLD   103;
      A     "PB_LAMP_ACK";
      =     L 0.2;
      BLD   103;
      CALL  "ALARM_BLOCK" (
           $1                       := L 0.0,
           $2                       := L 0.1,
           $3                       := L 0.2,
           $4                       := 5,
           $5                       := "fault_HS_22_06",
           $6                       := "fault_ack_HS_22_06",
           $7                       := DB110.DBX 1.6,
           $8                       := DB120.DBX 1.6,
           $9                       := DB100.DBW 28,
           $10                      := DB115.DBX 1.6);
      NOP   0;
NETWORK
TITLE =
      A     "check_HS_24_06";
      =     L 0.0;
      BLD   103;
      A     "1_second";
      =     L 0.1;
      BLD   103;
      A     "PB_LAMP_ACK";
      =     L 0.2;
      BLD   103;
      CALL  "ALARM_BLOCK" (
           $1                       := L 0.0,
           $2                       := L 0.1,
           $3                       := L 0.2,
           $4                       := 5,
           $5                       := "fault_HS_24_06",
           $6                       := "fault_ack_HS_24_06",
           $7                       := DB110.DBX 1.7,
           $8                       := DB120.DBX 1.7,
           $9                       := DB100.DBW 30,
           $10                      := DB115.DBX 1.7);
      NOP   0;
NETWORK
TITLE =
      A     "check_HS_24_07";
      =     L 0.0;
      BLD   103;
      A     "1_second";
      =     L 0.1;
      BLD   103;
      A     "PB_LAMP_ACK";
      =     L 0.2;
      BLD   103;
      CALL  "ALARM_BLOCK" (
           $1                       := L 0.0,
           $2                       := L 0.1,
           $3                       := L 0.2,
           $4                       := 5,
           $5                       := "fault_HS_24_07",
           $6                       := "fault_ack_HS_24_07",
           $7                       := DB110.DBX 0.0,
           $8                       := DB120.DBX 0.0,
           $9                       := DB100.DBW 0,
           $10                      := DB115.DBX 0.0);
      NOP   0;
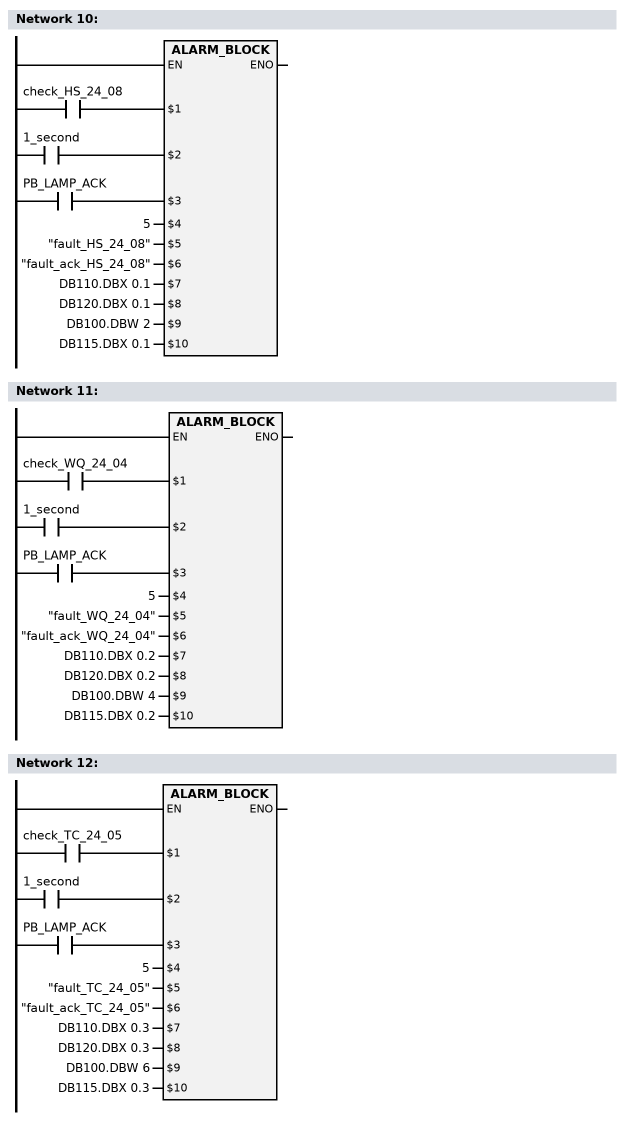
NETWORK
TITLE =
      A     "check_HS_24_08";
      =     L 0.0;
      BLD   103;
      A     "1_second";
      =     L 0.1;
      BLD   103;
      A     "PB_LAMP_ACK";
      =     L 0.2;
      BLD   103;
      CALL  "ALARM_BLOCK" (
           $1                       := L 0.0,
           $2                       := L 0.1,
           $3                       := L 0.2,
           $4                       := 5,
           $5                       := "fault_HS_24_08",
           $6                       := "fault_ack_HS_24_08",
           $7                       := DB110.DBX 0.1,
           $8                       := DB120.DBX 0.1,
           $9                       := DB100.DBW 2,
           $10                      := DB115.DBX 0.1);
      NOP   0;
NETWORK
TITLE =
      A     "check_WQ_24_04";
      =     L 0.0;
      BLD   103;
      A     "1_second";
      =     L 0.1;
      BLD   103;
      A     "PB_LAMP_ACK";
      =     L 0.2;
      BLD   103;
      CALL  "ALARM_BLOCK" (
           $1                       := L 0.0,
           $2                       := L 0.1,
           $3                       := L 0.2,
           $4                       := 5,
           $5                       := "fault_WQ_24_04",
           $6                       := "fault_ack_WQ_24_04",
           $7                       := DB110.DBX 0.2,
           $8                       := DB120.DBX 0.2,
           $9                       := DB100.DBW 4,
           $10                      := DB115.DBX 0.2);
      NOP   0;
NETWORK
TITLE =
      A     "check_TC_24_05";
      =     L 0.0;
      BLD   103;
      A     "1_second";
      =     L 0.1;
      BLD   103;
      A     "PB_LAMP_ACK";
      =     L 0.2;
      BLD   103;
      CALL  "ALARM_BLOCK" (
           $1                       := L 0.0,
           $2                       := L 0.1,
           $3                       := L 0.2,
           $4                       := 5,
           $5                       := "fault_TC_24_05",
           $6                       := "fault_ack_TC_24_05",
           $7                       := DB110.DBX 0.3,
           $8                       := DB120.DBX 0.3,
           $9                       := DB100.DBW 6,
           $10                      := DB115.DBX 0.3);
      NOP   0;
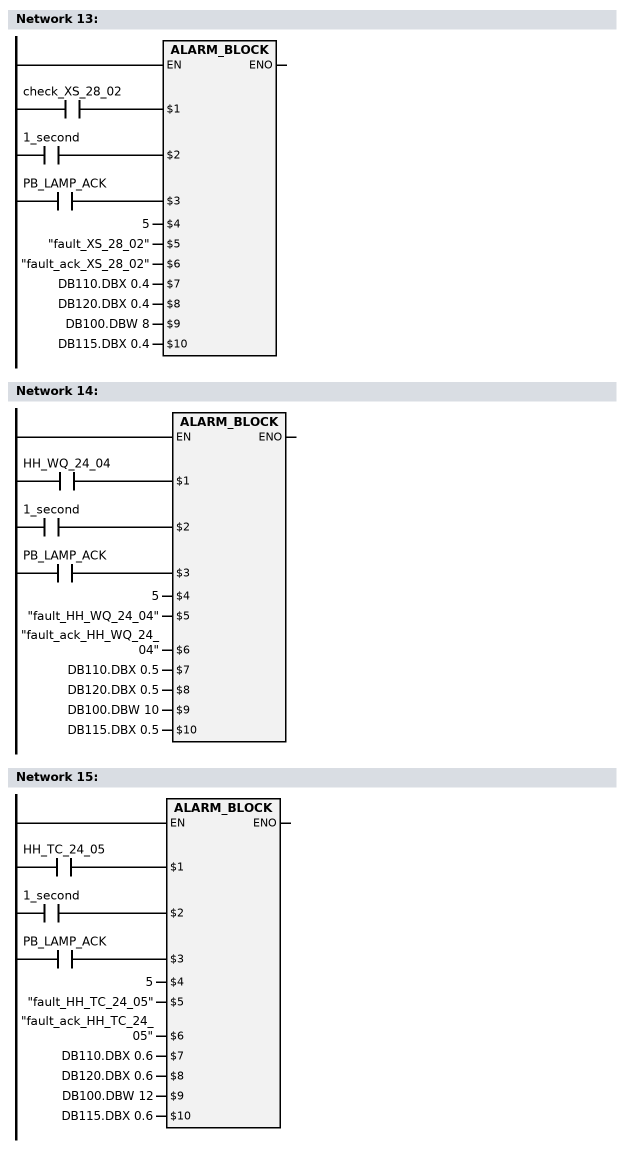
NETWORK
TITLE =
      A     "check_XS_28_02";
      =     L 0.0;
      BLD   103;
      A     "1_second";
      =     L 0.1;
      BLD   103;
      A     "PB_LAMP_ACK";
      =     L 0.2;
      BLD   103;
      CALL  "ALARM_BLOCK" (
           $1                       := L 0.0,
           $2                       := L 0.1,
           $3                       := L 0.2,
           $4                       := 5,
           $5                       := "fault_XS_28_02",
           $6                       := "fault_ack_XS_28_02",
           $7                       := DB110.DBX 0.4,
           $8                       := DB120.DBX 0.4,
           $9                       := DB100.DBW 8,
           $10                      := DB115.DBX 0.4);
      NOP   0;
NETWORK
TITLE =
      A     "HH_WQ_24_04";
      =     L 0.0;
      BLD   103;
      A     "1_second";
      =     L 0.1;
      BLD   103;
      A     "PB_LAMP_ACK";
      =     L 0.2;
      BLD   103;
      CALL  "ALARM_BLOCK" (
           $1                       := L 0.0,
           $2                       := L 0.1,
           $3                       := L 0.2,
           $4                       := 5,
           $5                       := "fault_HH_WQ_24_04",
           $6                       := "fault_ack_HH_WQ_24_04",
           $7                       := DB110.DBX 0.5,
           $8                       := DB120.DBX 0.5,
           $9                       := DB100.DBW 10,
           $10                      := DB115.DBX 0.5);
      NOP   0;
NETWORK
TITLE =
      A     "HH_TC_24_05";
      =     L 0.0;
      BLD   103;
      A     "1_second";
      =     L 0.1;
      BLD   103;
      A     "PB_LAMP_ACK";
      =     L 0.2;
      BLD   103;
      CALL  "ALARM_BLOCK" (
           $1                       := L 0.0,
           $2                       := L 0.1,
           $3                       := L 0.2,
           $4                       := 5,
           $5                       := "fault_HH_TC_24_05",
           $6                       := "fault_ack_HH_TC_24_05",
           $7                       := DB110.DBX 0.6,
           $8                       := DB120.DBX 0.6,
           $9                       := DB100.DBW 12,
           $10                      := DB115.DBX 0.6);
      NOP   0;
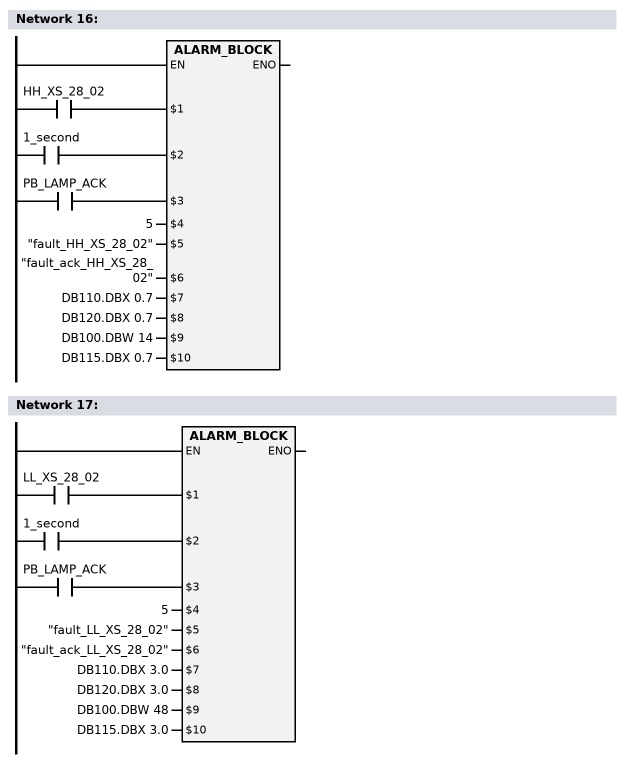
NETWORK
TITLE =
      A     "HH_XS_28_02";
      =     L 0.0;
      BLD   103;
      A     "1_second";
      =     L 0.1;
      BLD   103;
      A     "PB_LAMP_ACK";
      =     L 0.2;
      BLD   103;
      CALL  "ALARM_BLOCK" (
           $1                       := L 0.0,
           $2                       := L 0.1,
           $3                       := L 0.2,
           $4                       := 5,
           $5                       := "fault_HH_XS_28_02",
           $6                       := "fault_ack_HH_XS_28_02",
           $7                       := DB110.DBX 0.7,
           $8                       := DB120.DBX 0.7,
           $9                       := DB100.DBW 14,
           $10                      := DB115.DBX 0.7);
      NOP   0;
NETWORK
TITLE =
      A     "LL_XS_28_02";
      =     L 0.0;
      BLD   103;
      A     "1_second";
      =     L 0.1;
      BLD   103;
      A     "PB_LAMP_ACK";
      =     L 0.2;
      BLD   103;
      CALL  "ALARM_BLOCK" (
           $1                       := L 0.0,
           $2                       := L 0.1,
           $3                       := L 0.2,
           $4                       := 5,
           $5                       := "fault_LL_XS_28_02",
           $6                       := "fault_ack_LL_XS_28_02",
           $7                       := DB110.DBX 3.0,
           $8                       := DB120.DBX 3.0,
           $9                       := DB100.DBW 48,
           $10                      := DB115.DBX 3.0);
      NOP   0;
END_FUNCTION_BLOCK

FUNCTION_BLOCK "ALARM"	// FB 33
AUTHOR : GAW-LK
FAMILY : ALARM
NAME : ALARM
VERSION : 0.1
BEGIN
// (block stored without names or comments; labels and parameter names are numbered)
NETWORK
TITLE =
      L     DB110.DBW 0;
      L     0;
      ==I;
      =     L 1.0;
      L     DB110.DBW 2;
      L     0;
      ==I;
      =     L 1.1;
      L     DB110.DBW 4;
      L     0;
      ==I;
      =     L 1.2;
      L     DB110.DBW 6;
      L     0;
      ==I;
      =     L 1.3;
      L     DB110.DBW 8;
      L     0;
      ==I;
      =     L 1.4;
      L     DB110.DBW 10;
      L     0;
      ==I;
      =     L 1.5;
      L     DB110.DBW 12;
      L     0;
      ==I;
      =     L 1.6;
      L     DB110.DBW 14;
      L     0;
      ==I;
      =     L 1.7;
      L     DB110.DBW 16;
      L     0;
      ==I;
      =     L 2.0;
      ON    L 1.0;
      ON    L 1.1;
      ON    L 1.2;
      ON    L 1.3;
      ON    L 1.4;
      ON    L 1.5;
      ON    L 1.6;
      ON    L 1.7;
      ON    L 2.0;
      L     S5T#500MS;
      SD    T 5;
      A     T 5;
      =     L 100.0;
NETWORK
TITLE =
      L     DB110.DBW 0;
      L     DB120.DBW 0;
      ==I;
      =     L 4.0;
      L     DB110.DBW 2;
      L     DB120.DBW 2;
      ==I;
      =     L 4.1;
      L     DB110.DBW 4;
      L     DB120.DBW 4;
      ==I;
      =     L 4.2;
      L     DB110.DBW 6;
      L     DB120.DBW 6;
      ==I;
      =     L 4.3;
      L     DB110.DBW 8;
      L     DB120.DBW 8;
      ==I;
      =     L 4.4;
      L     DB110.DBW 10;
      L     DB120.DBW 10;
      ==I;
      =     L 4.5;
      L     DB110.DBW 12;
      L     DB120.DBW 12;
      ==I;
      =     L 4.6;
      L     DB110.DBW 14;
      L     DB120.DBW 14;
      ==I;
      =     L 4.7;
      L     DB110.DBW 16;
      L     DB120.DBW 16;
      ==I;
      =     L 5.0;
      ON    L 4.0;
      ON    L 4.1;
      ON    L 4.2;
      ON    L 4.3;
      ON    L 4.4;
      ON    L 4.5;
      ON    L 4.6;
      ON    L 4.7;
      ON    L 5.0;
      L     S5T#500MS;
      SD    T 6;
      O     T 6;
      O     "AlarmOnEnzym";
      =     "XA28_01_ON";
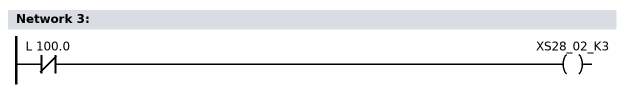
NETWORK
TITLE =
      AN    L 100.0;
      =     "XS28_02_K3";
END_FUNCTION_BLOCK

FUNCTION_BLOCK "Batch"	// FB 90
VERSION : 0.1
BEGIN
// (block stored without names or comments; labels and parameter names are numbered)
NETWORK
TITLE =
      TAR1  LD 4;
NETWORK
TITLE =
      A     DIX [AR2,P#0.0];
      AN    DIX [AR2,P#16.0];
      =     DIX [AR2,P#738.1];
      =     DIX [AR2,P#16.1];
      S     DIX [AR2,P#16.0];
      A     DIX [AR2,P#14.1];
      S     DIX [AR2,P#734.0];
      A     DIX [AR2,P#734.0];
      R     DIX [AR2,P#16.0];
      L     DIW [AR2,P#740.0];
      T     DIW [AR2,P#18.0];
      O     DIX [AR2,P#738.1];
      O     DIX [AR2,P#734.0];
      JC    M023;
      A     DIX [AR2,P#16.0];
      JC    M001;
      BEU;
M001: NOP   0;
      SET;
      R     L 22.0;
      AN    DIX [AR2,P#738.0];
      JC    M002;
      R     DIX [AR2,P#738.0];
      L     DIW [AR2,P#736.0];
      L     1;
      +I;
      T     DIW [AR2,P#736.0];
      L     DIW [AR2,P#10.0];
      >=I;
      =     DIX [AR2,P#734.0];
      JC    M027;
M002: NOP   0;
      LAR1  P#DIX 20.0;
      L     0;
      T     LW 8;
M003: L     DIW [AR2,P#736.0];
      L     LW 8;
      ==I;
      JC    M004;
      L     DIW [AR2,P#736.0];
      L     272;
      *I;
      +AR1;
      L     LW 8;
      L     1;
      +I;
      T     LW 8;
      TAR1  LD 16;
      LOOP  M003;
M004: NOP   0;
      SET;
      R      [AR1,P#32.2];
      L     0;
      L     W [AR1,P#20.0];
      ==I;
      JC    M008;
      L     1;
      L     W [AR1,P#20.0];
      ==I;
      JC    M009;
      L     2;
      L     W [AR1,P#20.0];
      ==I;
      JC    M005;
      L     3;
      L     W [AR1,P#20.0];
      ==I;
      JC    M006;
      JU    M007;
M005: S      [AR1,P#32.0];
      SET;
      =      [AR1,P#32.3];
      A      [AR1,P#32.3];
      A      [AR1,P#32.4];
      JC    M016;
      JU    M018;
M006: A      [AR1,P#32.0];
      JC    M015;
      L     L#0;
      T     DID [AR2,P#742.0];
      SET;
      S      [AR1,P#32.0];
      JU    M015;
M007: NOP   0;
M008: L     DID [AR2,P#2.0];
      JU    M013;
M009: SET;
      =     L 22.0;
      L     W [AR1,P#30.0];
      L     1;
      -I;
      L     DIW [AR2,P#736.0];
      -I;
      T     LW 20;
      L     0;
      >I;
      JC    M010;
      JU    M012;
M010: LAR1  LD 16;
      L     LW 20;
      L     272;
      *I;
      +AR1;
      L     DID [AR2,P#2.0];
      T     D [AR1,P#16.0];
      A      [AR1,P#32.0];
      JC    M011;
      L     D [AR1,P#16.0];
      T     D [AR1,P#12.0];
      L     0.000000e+00;
      T     D [AR1,P#4.0];
      SET;
      S      [AR1,P#32.2];
      S      [AR1,P#32.0];
M011: L     D [AR1,P#16.0];
      L     D [AR1,P#12.0];
      -R;
      L     D [AR1,P#4.0];
      +R;
      T     D [AR1,P#4.0];
      L     D [AR1,P#16.0];
      T     D [AR1,P#12.0];
      LAR1  LD 16;
M012: L     DID [AR2,P#6.0];
      JU    M013;
M013: T     D [AR1,P#16.0];
      A      [AR1,P#32.0];
      JC    M014;
      L     0.000000e+00;
      T     D [AR1,P#4.0];
      T     D [AR1,P#12.0];
      L     L#0;
      T     DID [AR2,P#742.0];
      A     L 22.0;
      JC    M014;
      L     D [AR1,P#16.0];
      T     D [AR1,P#12.0];
M014: L     D [AR1,P#16.0];
      L     D [AR1,P#12.0];
      -R;
      L     D [AR1,P#4.0];
      +R;
      T     D [AR1,P#4.0];
      L     D [AR1,P#16.0];
      T     D [AR1,P#12.0];
      L     D [AR1,P#0.0];
      L     D [AR1,P#8.0];
      -R;
      L     D [AR1,P#4.0];
      >R;
      =     L 10.0;
      SET;
      S      [AR1,P#32.0];
      A     L 10.0;
      AN     [AR1,P#32.2];
      =      [AR1,P#32.1];
      A     L 10.0;
      JC    M017;
M015: L     3;
      L     W [AR1,P#20.0];
      ==I;
      A     DIX [AR2,P#14.0];
      JC    M018;
      L     DIW [AR2,P#12.0];
      L     DID [AR2,P#742.0];
      +D;
      T     DID [AR2,P#742.0];
      L     1000;
      /D;
      T     D [AR1,P#26.0];
      L     D [AR1,P#22.0];
      >=D;
M016: S     DIX [AR2,P#738.0];
      R      [AR1,P#32.0];
      JU    M018;
M017: L     0;
      T     DID [AR2,P#742.0];
M018: NOP   0;
      L     0;
      T     LW 24;
      T     DIW [AR2,P#740.0];
M019: LAR1  P#DIX 20.0;
      L     LW 24;
      L     272;
      *I;
      +AR1;
      AN     [AR1,P#32.0];
      JC    M020;
      L     LW 24;
      L     1;
      SLW;
      L     DIW [AR2,P#740.0];
      +I;
      T     DIW [AR2,P#740.0];
      JU    M021;
M020: L     LW 24;
      L     0;
      SLW;
      L     DIW [AR2,P#740.0];
      +I;
      T     DIW [AR2,P#740.0];
M021: L     1;
      L     LW 24;
      +I;
      T     LW 24;
      L     DIW [AR2,P#10.0];
      >=I;
      JC    M022;
      LOOP  M019;
M022: JU    M027;
M023: L     0;
      T     LW 24;
      T     DIW [AR2,P#740.0];
M024: LAR1  P#DIX 20.0;
      L     LW 24;
      L     272;
      *I;
      +AR1;
      A     DIX [AR2,P#734.0];
      JC    M025;
      L     0.000000e+00;
      T     D [AR1,P#16.0];
      T     D [AR1,P#12.0];
      T     D [AR1,P#4.0];
      L     L#0;
      T     D [AR1,P#26.0];
      L     0;
      T     W [AR1,P#26.0];
M025: SET;
      R      [AR1,P#32.0];
      R      [AR1,P#32.2];
      R      [AR1,P#32.1];
      R      [AR1,P#32.3];
      R      [AR1,P#32.4];
      L     1;
      L     LW 24;
      +I;
      T     LW 24;
      L     DIW [AR2,P#10.0];
      >=I;
      JC    M026;
      LOOP  M024;
M026: A     DIX [AR2,P#734.0];
      R     DIX [AR2,P#734.0];
      L     0;
      T     DIW [AR2,P#736.0];
      T     DIW [AR2,P#740.0];
NETWORK
TITLE =
M027: LAR1  LD 4;
END_FUNCTION_BLOCK

FUNCTION "BatchControl" : VOID	// FC 10
VERSION : 0.1
BEGIN
// (block stored without names or comments; labels and parameter names are numbered)
NETWORK
TITLE =
      CALL  "RecipeControl" (
           $1                       := "Batch_Starch_Started",
           $2                       := P#DB90.DBX 0.0,
           $3                       := P#DB91.DBX 0.0);
NETWORK
TITLE =
      CALL  "Batch" , "DataBatchControl" (
           DIX 0.0                  := "IMP_START_STARCH",
           DID 2                    := "WQ_24_04_Value",
           DID 6                    := "TC_24_05_Value",
           DIW 10                   := 14,
           DIW 12                   := "Cycle_Time",
           DIX 14.0                 := "Hold_Mixing_Time_Starch",
           DIX 14.1                 := DB30.DBX 0.6,
           DIX 16.0                 := "Batch_Starch_Running",
           DIX 16.1                 := "Batch_Starch_Started",
           DIW 18                   := DB91.DBW 90);
NETWORK
TITLE =
      A     DB30.DBX 0.6;
      R     DB30.DBX 0.6;
NETWORK
TITLE =
      CALL  "DosLine" (
           $1                       := DB91.DBD 36,
           $2                       := DB91.DBD 82,
           $3                       := L#5,
           $4                       := 0,
           $5                       := 0,
           $6                       := FALSE,
           $7                       := DB91.DBD 40,
           $8                       := P#L 4.0,
           $9                       := P#L 8.0,
           $10                      := P#L 8.0,
           $11                      := "Dos_On_Water_Starch",
           $12                      := P#DB92.DBX 20.0);
NETWORK
TITLE =
      CALL  "DosLine" (
           $1                       := L#0,
           $2                       := L#0,
           $3                       := L#0,
           $4                       := 2,
           $5                       := 0,
           $6                       := "M24_01_RUN",
           $7                       := P#L 10.0,
           $8                       := P#L 4.0,
           $9                       := "Cmd_Agitator_On_Starch",
           $10                      := P#L 8.0,
           $11                      := P#L 8.0,
           $12                      := P#DB92.DBX 54.0);
NETWORK
TITLE =
      CALL  "DosLine" (
           $1                       := DB91.DBD 44,
           $2                       := DB91.DBD 78,
           $3                       := L#1,
           $4                       := 0,
           $5                       := 0,
           $6                       := FALSE,
           $7                       := DB91.DBD 48,
           $8                       := P#L 4.0,
           $9                       := P#L 8.0,
           $10                      := P#L 8.0,
           $11                      := "Dos_On_Powder_Starch",
           $12                      := P#DB92.DBX 88.0);
NETWORK
TITLE =
      L     DB91.DBW 8;
      T     LD 0;
      CALL  "DosLine" (
           $1                       := L#0,
           $2                       := L#0,
           $3                       := P#L 0.0,
           $4                       := 3,
           $5                       := 0,
           $6                       := FALSE,
           $7                       := P#L 10.0,
           $8                       := P#L 0.0,
           $9                       := P#L 8.0,
           $10                      := P#L 8.0,
           $11                      := P#L 8.0,
           $12                      := P#DB92.DBX 122.0);
      L     LD 0;
      T     DB91.DBW 10;
NETWORK
TITLE =
      CALL  "DosLine" (
           $1                       := L#0,
           $2                       := L#0,
           $3                       := L#0,
           $4                       := 2,
           $5                       := 0,
           $6                       := "Enzyme_Done_Starch",
           $7                       := P#L 10.0,
           $8                       := P#L 4.0,
           $9                       := "Cmd_Enzym_On_Starch",
           $10                      := P#L 8.0,
           $11                      := P#L 8.0,
           $12                      := P#DB92.DBX 156.0);
NETWORK
TITLE =
      A     DB30.DBX 10.0;
      JC    M001;
      L     DB91.DBD 92;
      T     LD 14;
      L     DB91.DBD 86;
      T     LD 18;
      L     L#20;
      T     LD 22;
      L     10;
      T     LW 26;
      JU    M002;
M001: L     0.000000e+00;
      T     LD 14;
      T     LD 14;
      T     LD 18;
      L     0;
      T     LD 22;
M002: T     LW 26;
NETWORK
TITLE =
      CALL  "DosLine" (
           $1                       := P#L 14.0,
           $2                       := P#L 18.0,
           $3                       := P#L 22.0,
           $4                       := 1,
           $5                       := P#L 26.0,
           $6                       := FALSE,
           $7                       := P#L 28.0,
           $8                       := P#L 4.0,
           $9                       := P#L 8.0,
           $10                      := P#L 8.0,
           $11                      := "Dos_On_EnzSteam_Starch",
           $12                      := P#DB92.DBX 190.0);
NETWORK
TITLE =
      L     0.000000e+00;
      A     DB30.DBX 10.0;
      JC    M003;
      L     LD 28;
M003: T     DB91.DBD 96;
NETWORK
TITLE =
      L     L#0;
      A     DB30.DBX 10.0;
      JC    M004;
      L     DB91.DBW 100;
M004: T     LD 0;
      CALL  "DosLine" (
           $1                       := L#0,
           $2                       := L#0,
           $3                       := P#L 0.0,
           $4                       := 3,
           $5                       := 0,
           $6                       := FALSE,
           $7                       := P#L 10.0,
           $8                       := P#L 0.0,
           $9                       := P#L 8.0,
           $10                      := "Active_Hold_Temp_Starch",
           $11                      := P#L 8.0,
           $12                      := P#DB92.DBX 224.0);
      L     LD 0;
      T     DB91.DBW 102;
NETWORK
TITLE =
      CALL  "DosLine" (
           $1                       := DB91.DBD 52,
           $2                       := DB91.DBD 86,
           $3                       := L#20,
           $4                       := 1,
           $5                       := 10,
           $6                       := FALSE,
           $7                       := DB91.DBD 56,
           $8                       := P#L 4.0,
           $9                       := P#L 8.0,
           $10                      := P#L 8.0,
           $11                      := "Dos_On_Steam_Starch",
           $12                      := P#DB92.DBX 258.0);
NETWORK
TITLE =
      L     DB91.DBW 12;
      T     LD 0;
      CALL  "DosLine" (
           $1                       := L#0,
           $2                       := L#0,
           $3                       := P#L 0.0,
           $4                       := 3,
           $5                       := 0,
           $6                       := FALSE,
           $7                       := P#L 10.0,
           $8                       := P#L 0.0,
           $9                       := P#L 8.0,
           $10                      := "Active_Temp_Starch",
           $11                      := P#L 8.0,
           $12                      := P#DB92.DBX 292.0);
      L     LD 0;
      T     DB91.DBW 14;
NETWORK
TITLE =
      CALL  "DosLine" (
           $1                       := DB91.DBD 60,
           $2                       := DB91.DBD 82,
           $3                       := L#5,
           $4                       := 0,
           $5                       := 0,
           $6                       := FALSE,
           $7                       := DB91.DBD 64,
           $8                       := P#L 4.0,
           $9                       := P#L 8.0,
           $10                      := "Active_Dil_Water_Starch",
           $11                      := "Dos_On_Dil_Water_Starch",
           $12                      := P#DB92.DBX 326.0);
NETWORK
TITLE =
      L     DB91.DBW 16;
      T     LD 0;
      CALL  "DosLine" (
           $1                       := L#0,
           $2                       := L#0,
           $3                       := P#L 0.0,
           $4                       := 3,
           $5                       := 0,
           $6                       := FALSE,
           $7                       := P#L 10.0,
           $8                       := P#L 0.0,
           $9                       := P#L 8.0,
           $10                      := P#L 8.0,
           $11                      := P#L 8.0,
           $12                      := P#DB92.DBX 360.0);
      L     LD 0;
      T     DB91.DBW 18;
NETWORK
TITLE =
      CALL  "DosLine" (
           $1                       := L#0,
           $2                       := L#0,
           $3                       := L#0,
           $4                       := 2,
           $5                       := 0,
           $6                       := "Discharged1_Starch",
           $7                       := P#L 10.0,
           $8                       := P#L 4.0,
           $9                       := "Cmd_Discharge1_On_Starch",
           $10                      := "Active_Discharge1_Starch",
           $11                      := P#L 8.0,
           $12                      := P#DB92.DBX 394.0);
NETWORK
TITLE =
      CALL  "DosLine" (
           $1                       := DB91.DBD 68,
           $2                       := DB91.DBD 82,
           $3                       := L#5,
           $4                       := 0,
           $5                       := 0,
           $6                       := FALSE,
           $7                       := DB91.DBD 72,
           $8                       := P#L 4.0,
           $9                       := P#L 8.0,
           $10                      := P#L 8.0,
           $11                      := "Dos_On_Flushwater_Starch",
           $12                      := P#DB92.DBX 428.0);
NETWORK
TITLE =
      CALL  "DosLine" (
           $1                       := L#0,
           $2                       := L#0,
           $3                       := L#0,
           $4                       := 2,
           $5                       := 0,
           $6                       := "Discharged2_Starch",
           $7                       := P#L 10.0,
           $8                       := P#L 4.0,
           $9                       := "Cmd_Discharge2_On_Starch",
           $10                      := "Active_Discharge2_Starch",
           $11                      := P#L 8.0,
           $12                      := P#DB92.DBX 462.0);
END_FUNCTION

FUNCTION "RecipeControl" : VOID	// FC 90
VERSION : 0.1
BEGIN
// (block stored without names or comments; labels and parameter names are numbered)
NETWORK
TITLE =
      BLD   5;
      T     LD 18;
      TAK;
      T     LD 22;
      L     P##PARAM2;
      LAR1;
      L     W [AR1,P#0.0];
      T     LW 16;
      OPN   DB [LW 16];
      L     D [AR1,P#2.0];
      LAR1;
      L     LD 22;
      L     LD 18;
      L     D [AR1,P#0.0];
      L     0;
      >R;
      JC    M001;
      BEU;
M001: BLD   5;
      T     LD 18;
      TAK;
      T     LD 22;
      L     P##PARAM2;
      LAR1;
      L     W [AR1,P#0.0];
      T     LW 16;
      OPN   DB [LW 16];
      L     D [AR1,P#2.0];
      LAR1;
      L     LD 22;
      L     LD 18;
      L     D [AR1,P#4.0];
      L     0;
      >R;
      JC    M002;
      BEU;
M002: BLD   5;
      T     LD 18;
      TAK;
      T     LD 22;
      L     P##PARAM2;
      LAR1;
      L     W [AR1,P#0.0];
      T     LW 16;
      OPN   DB [LW 16];
      L     D [AR1,P#2.0];
      LAR1;
      L     LD 22;
      L     LD 18;
      L     D [AR1,P#28.0];
      L     0;
      >R;
      JC    M003;
      BEU;
M003: BLD   5;
      T     LD 18;
      TAK;
      T     LD 22;
      L     P##PARAM2;
      LAR1;
      L     W [AR1,P#0.0];
      T     LW 16;
      OPN   DB [LW 16];
      L     D [AR1,P#2.0];
      LAR1;
      L     LD 22;
      L     LD 18;
      L     D [AR1,P#28.0];
      BLD   5;
      T     LD 18;
      TAK;
      T     LD 22;
      L     P##PARAM2;
      LAR1;
      L     W [AR1,P#0.0];
      T     LW 16;
      OPN   DB [LW 16];
      L     D [AR1,P#2.0];
      LAR1;
      L     LD 22;
      L     LD 18;
      L     D [AR1,P#4.0];
      -R;
      BLD   5;
      T     LD 18;
      TAK;
      T     LD 22;
      L     P##PARAM2;
      LAR1;
      L     W [AR1,P#0.0];
      T     LW 16;
      OPN   DB [LW 16];
      L     D [AR1,P#2.0];
      LAR1;
      L     LD 22;
      L     LD 18;
      L     D [AR1,P#4.0];
      /R;
      T     LD 0;
      BLD   5;
      T     LD 18;
      TAK;
      T     LD 22;
      L     P##PARAM2;
      LAR1;
      L     W [AR1,P#0.0];
      T     LW 16;
      OPN   DB [LW 16];
      L     D [AR1,P#2.0];
      LAR1;
      L     LD 22;
      L     LD 18;
      L     D [AR1,P#0.0];
      L     LD 0;
      *R;
      T     LD 4;
      BLD   5;
      T     LD 18;
      TAK;
      T     LD 22;
      L     P##PARAM2;
      LAR1;
      L     W [AR1,P#0.0];
      T     LW 16;
      OPN   DB [LW 16];
      L     D [AR1,P#2.0];
      LAR1;
      L     LD 22;
      L     LD 18;
      L     D [AR1,P#0.0];
      +R;
      T     LD 8;
      BLD   5;
      T     LD 18;
      TAK;
      T     LD 22;
      L     P##PARAM2;
      LAR1;
      L     W [AR1,P#0.0];
      T     LW 16;
      OPN   DB [LW 16];
      L     D [AR1,P#2.0];
      LAR1;
      L     LD 22;
      L     LD 18;
      L     D [AR1,P#0.0];
      /R;
      T     LD 12;
      BLD   5;
      T     LD 18;
      TAK;
      T     LD 22;
      L     P##PARAM2;
      LAR1;
      L     W [AR1,P#0.0];
      T     LW 16;
      OPN   DB [LW 16];
      L     D [AR1,P#2.0];
      LAR1;
      L     LD 22;
      L     LD 18;
      L     D [AR1,P#0.0];
      L     LD 12;
      /R;
      BLD   5;
      T     LD 18;
      TAK;
      T     LD 22;
      L     P##PARAM2;
      LAR1;
      L     W [AR1,P#0.0];
      T     LW 16;
      OPN   DB [LW 16];
      L     D [AR1,P#2.0];
      LAR1;
      L     LD 22;
      L     LD 18;
      T     D [AR1,P#44.0];
      L     LD 4;
      L     LD 12;
      /R;
      BLD   5;
      T     LD 18;
      TAK;
      T     LD 22;
      L     P##PARAM2;
      LAR1;
      L     W [AR1,P#0.0];
      T     LW 16;
      OPN   DB [LW 16];
      L     D [AR1,P#2.0];
      LAR1;
      L     LD 22;
      L     LD 18;
      L     D [AR1,P#68.0];
      -R;
      BLD   5;
      T     LD 18;
      TAK;
      T     LD 22;
      L     P##PARAM2;
      LAR1;
      L     W [AR1,P#0.0];
      T     LW 16;
      OPN   DB [LW 16];
      L     D [AR1,P#2.0];
      LAR1;
      L     LD 22;
      L     LD 18;
      L     D [AR1,P#60.0];
      -R;
      BLD   5;
      T     LD 18;
      TAK;
      T     LD 22;
      L     P##PARAM2;
      LAR1;
      L     W [AR1,P#0.0];
      T     LW 16;
      OPN   DB [LW 16];
      L     D [AR1,P#2.0];
      LAR1;
      L     LD 22;
      L     LD 18;
      T     D [AR1,P#36.0];
NETWORK
TITLE =
      AN    #PARAM1;
      BEC;
      BLD   5;
      T     LD 18;
      TAK;
      T     LD 22;
      L     P##PARAM2;
      LAR1;
      L     W [AR1,P#0.0];
      T     LW 16;
      OPN   DB [LW 16];
      L     D [AR1,P#2.0];
      LAR1;
      L     LD 22;
      L     LD 18;
      L     D [AR1,P#0.0];
      BLD   5;
      T     LD 18;
      TAK;
      T     LD 22;
      L     P##PARAM3;
      LAR1;
      L     W [AR1,P#0.0];
      T     LW 16;
      OPN   DB [LW 16];
      L     D [AR1,P#2.0];
      LAR1;
      L     LD 22;
      L     LD 18;
      T     D [AR1,P#0.0];
      BLD   5;
      T     LD 18;
      TAK;
      T     LD 22;
      L     P##PARAM2;
      LAR1;
      L     W [AR1,P#0.0];
      T     LW 16;
      OPN   DB [LW 16];
      L     D [AR1,P#2.0];
      LAR1;
      L     LD 22;
      L     LD 18;
      L     D [AR1,P#4.0];
      BLD   5;
      T     LD 18;
      TAK;
      T     LD 22;
      L     P##PARAM3;
      LAR1;
      L     W [AR1,P#0.0];
      T     LW 16;
      OPN   DB [LW 16];
      L     D [AR1,P#2.0];
      LAR1;
      L     LD 22;
      L     LD 18;
      T     D [AR1,P#4.0];
      BLD   5;
      T     LD 18;
      TAK;
      T     LD 22;
      L     P##PARAM2;
      LAR1;
      L     W [AR1,P#0.0];
      T     LW 16;
      OPN   DB [LW 16];
      L     D [AR1,P#2.0];
      LAR1;
      L     LD 22;
      L     LD 18;
      L     D [AR1,P#36.0];
      BLD   5;
      T     LD 18;
      TAK;
      T     LD 22;
      L     P##PARAM3;
      LAR1;
      L     W [AR1,P#0.0];
      T     LW 16;
      OPN   DB [LW 16];
      L     D [AR1,P#2.0];
      LAR1;
      L     LD 22;
      L     LD 18;
      T     D [AR1,P#36.0];
      BLD   5;
      T     LD 18;
      TAK;
      T     LD 22;
      L     P##PARAM2;
      LAR1;
      L     W [AR1,P#0.0];
      T     LW 16;
      OPN   DB [LW 16];
      L     D [AR1,P#2.0];
      LAR1;
      L     LD 22;
      L     LD 18;
      L     D [AR1,P#44.0];
      BLD   5;
      T     LD 18;
      TAK;
      T     LD 22;
      L     P##PARAM3;
      LAR1;
      L     W [AR1,P#0.0];
      T     LW 16;
      OPN   DB [LW 16];
      L     D [AR1,P#2.0];
      LAR1;
      L     LD 22;
      L     LD 18;
      T     D [AR1,P#44.0];
      BLD   5;
      T     LD 18;
      TAK;
      T     LD 22;
      L     P##PARAM2;
      LAR1;
      L     W [AR1,P#0.0];
      T     LW 16;
      OPN   DB [LW 16];
      L     D [AR1,P#2.0];
      LAR1;
      L     LD 22;
      L     LD 18;
      L     W [AR1,P#8.0];
      BLD   5;
      T     LD 18;
      TAK;
      T     LD 22;
      L     P##PARAM3;
      LAR1;
      L     W [AR1,P#0.0];
      T     LW 16;
      OPN   DB [LW 16];
      L     D [AR1,P#2.0];
      LAR1;
      L     LD 22;
      L     LD 18;
      T     W [AR1,P#8.0];
      BLD   5;
      T     LD 18;
      TAK;
      T     LD 22;
      L     P##PARAM2;
      LAR1;
      L     W [AR1,P#0.0];
      T     LW 16;
      OPN   DB [LW 16];
      L     D [AR1,P#2.0];
      LAR1;
      L     LD 22;
      L     LD 18;
      L     D [AR1,P#52.0];
      BLD   5;
      T     LD 18;
      TAK;
      T     LD 22;
      L     P##PARAM3;
      LAR1;
      L     W [AR1,P#0.0];
      T     LW 16;
      OPN   DB [LW 16];
      L     D [AR1,P#2.0];
      LAR1;
      L     LD 22;
      L     LD 18;
      T     D [AR1,P#52.0];
      BLD   5;
      T     LD 18;
      TAK;
      T     LD 22;
      L     P##PARAM2;
      LAR1;
      L     W [AR1,P#0.0];
      T     LW 16;
      OPN   DB [LW 16];
      L     D [AR1,P#2.0];
      LAR1;
      L     LD 22;
      L     LD 18;
      L     W [AR1,P#12.0];
      BLD   5;
      T     LD 18;
      TAK;
      T     LD 22;
      L     P##PARAM3;
      LAR1;
      L     W [AR1,P#0.0];
      T     LW 16;
      OPN   DB [LW 16];
      L     D [AR1,P#2.0];
      LAR1;
      L     LD 22;
      L     LD 18;
      T     W [AR1,P#12.0];
      BLD   5;
      T     LD 18;
      TAK;
      T     LD 22;
      L     P##PARAM2;
      LAR1;
      L     W [AR1,P#0.0];
      T     LW 16;
      OPN   DB [LW 16];
      L     D [AR1,P#2.0];
      LAR1;
      L     LD 22;
      L     LD 18;
      L     D [AR1,P#60.0];
      BLD   5;
      T     LD 18;
      TAK;
      T     LD 22;
      L     P##PARAM3;
      LAR1;
      L     W [AR1,P#0.0];
      T     LW 16;
      OPN   DB [LW 16];
      L     D [AR1,P#2.0];
      LAR1;
      L     LD 22;
      L     LD 18;
      T     D [AR1,P#60.0];
      BLD   5;
      T     LD 18;
      TAK;
      T     LD 22;
      L     P##PARAM2;
      LAR1;
      L     W [AR1,P#0.0];
      T     LW 16;
      OPN   DB [LW 16];
      L     D [AR1,P#2.0];
      LAR1;
      L     LD 22;
      L     LD 18;
      L     W [AR1,P#16.0];
      BLD   5;
      T     LD 18;
      TAK;
      T     LD 22;
      L     P##PARAM3;
      LAR1;
      L     W [AR1,P#0.0];
      T     LW 16;
      OPN   DB [LW 16];
      L     D [AR1,P#2.0];
      LAR1;
      L     LD 22;
      L     LD 18;
      T     W [AR1,P#16.0];
      BLD   5;
      T     LD 18;
      TAK;
      T     LD 22;
      L     P##PARAM2;
      LAR1;
      L     W [AR1,P#0.0];
      T     LW 16;
      OPN   DB [LW 16];
      L     D [AR1,P#2.0];
      LAR1;
      L     LD 22;
      L     LD 18;
      L     W [AR1,P#20.0];
      BLD   5;
      T     LD 18;
      TAK;
      T     LD 22;
      L     P##PARAM3;
      LAR1;
      L     W [AR1,P#0.0];
      T     LW 16;
      OPN   DB [LW 16];
      L     D [AR1,P#2.0];
      LAR1;
      L     LD 22;
      L     LD 18;
      T     W [AR1,P#20.0];
      BLD   5;
      T     LD 18;
      TAK;
      T     LD 22;
      L     P##PARAM2;
      LAR1;
      L     W [AR1,P#0.0];
      T     LW 16;
      OPN   DB [LW 16];
      L     D [AR1,P#2.0];
      LAR1;
      L     LD 22;
      L     LD 18;
      L     D [AR1,P#68.0];
      BLD   5;
      T     LD 18;
      TAK;
      T     LD 22;
      L     P##PARAM3;
      LAR1;
      L     W [AR1,P#0.0];
      T     LW 16;
      OPN   DB [LW 16];
      L     D [AR1,P#2.0];
      LAR1;
      L     LD 22;
      L     LD 18;
      T     D [AR1,P#68.0];
      BLD   5;
      T     LD 18;
      TAK;
      T     LD 22;
      L     P##PARAM2;
      LAR1;
      L     W [AR1,P#0.0];
      T     LW 16;
      OPN   DB [LW 16];
      L     D [AR1,P#2.0];
      LAR1;
      L     LD 22;
      L     LD 18;
      L     W [AR1,P#24.0];
      BLD   5;
      T     LD 18;
      TAK;
      T     LD 22;
      L     P##PARAM3;
      LAR1;
      L     W [AR1,P#0.0];
      T     LW 16;
      OPN   DB [LW 16];
      L     D [AR1,P#2.0];
      LAR1;
      L     LD 22;
      L     LD 18;
      T     W [AR1,P#24.0];
      BLD   5;
      T     LD 18;
      TAK;
      T     LD 22;
      L     P##PARAM2;
      LAR1;
      L     W [AR1,P#0.0];
      T     LW 16;
      OPN   DB [LW 16];
      L     D [AR1,P#2.0];
      LAR1;
      L     LD 22;
      L     LD 18;
      L     D [AR1,P#78.0];
      BLD   5;
      T     LD 18;
      TAK;
      T     LD 22;
      L     P##PARAM3;
      LAR1;
      L     W [AR1,P#0.0];
      T     LW 16;
      OPN   DB [LW 16];
      L     D [AR1,P#2.0];
      LAR1;
      L     LD 22;
      L     LD 18;
      T     D [AR1,P#78.0];
      BLD   5;
      T     LD 18;
      TAK;
      T     LD 22;
      L     P##PARAM2;
      LAR1;
      L     W [AR1,P#0.0];
      T     LW 16;
      OPN   DB [LW 16];
      L     D [AR1,P#2.0];
      LAR1;
      L     LD 22;
      L     LD 18;
      L     D [AR1,P#82.0];
      BLD   5;
      T     LD 18;
      TAK;
      T     LD 22;
      L     P##PARAM3;
      LAR1;
      L     W [AR1,P#0.0];
      T     LW 16;
      OPN   DB [LW 16];
      L     D [AR1,P#2.0];
      LAR1;
      L     LD 22;
      L     LD 18;
      T     D [AR1,P#82.0];
      BLD   5;
      T     LD 18;
      TAK;
      T     LD 22;
      L     P##PARAM2;
      LAR1;
      L     W [AR1,P#0.0];
      T     LW 16;
      OPN   DB [LW 16];
      L     D [AR1,P#2.0];
      LAR1;
      L     LD 22;
      L     LD 18;
      L     D [AR1,P#86.0];
      BLD   5;
      T     LD 18;
      TAK;
      T     LD 22;
      L     P##PARAM3;
      LAR1;
      L     W [AR1,P#0.0];
      T     LW 16;
      OPN   DB [LW 16];
      L     D [AR1,P#2.0];
      LAR1;
      L     LD 22;
      L     LD 18;
      T     D [AR1,P#86.0];
      A     DB30.DBX 10.0;
      JC    M004;
      BLD   5;
      T     LD 18;
      TAK;
      T     LD 22;
      L     P##PARAM2;
      LAR1;
      L     W [AR1,P#0.0];
      T     LW 16;
      OPN   DB [LW 16];
      L     D [AR1,P#2.0];
      LAR1;
      L     LD 22;
      L     LD 18;
      L     D [AR1,P#92.0];
      BLD   5;
      T     LD 18;
      TAK;
      T     LD 22;
      L     P##PARAM3;
      LAR1;
      L     W [AR1,P#0.0];
      T     LW 16;
      OPN   DB [LW 16];
      L     D [AR1,P#2.0];
      LAR1;
      L     LD 22;
      L     LD 18;
      T     D [AR1,P#92.0];
      BLD   5;
      T     LD 18;
      TAK;
      T     LD 22;
      L     P##PARAM2;
      LAR1;
      L     W [AR1,P#0.0];
      T     LW 16;
      OPN   DB [LW 16];
      L     D [AR1,P#2.0];
      LAR1;
      L     LD 22;
      L     LD 18;
      L     W [AR1,P#100.0];
      BLD   5;
      T     LD 18;
      TAK;
      T     LD 22;
      L     P##PARAM3;
      LAR1;
      L     W [AR1,P#0.0];
      T     LW 16;
      OPN   DB [LW 16];
      L     D [AR1,P#2.0];
      LAR1;
      L     LD 22;
      L     LD 18;
      T     W [AR1,P#100.0];
      BEU;
M004: L     0.000000e+00;
      BLD   5;
      T     LD 18;
      TAK;
      T     LD 22;
      L     P##PARAM3;
      LAR1;
      L     W [AR1,P#0.0];
      T     LW 16;
      OPN   DB [LW 16];
      L     D [AR1,P#2.0];
      LAR1;
      L     LD 22;
      L     LD 18;
      T     D [AR1,P#92.0];
      BLD   5;
      T     LD 18;
      TAK;
      T     LD 22;
      L     P##PARAM3;
      LAR1;
      L     W [AR1,P#0.0];
      T     LW 16;
      OPN   DB [LW 16];
      L     D [AR1,P#2.0];
      LAR1;
      L     LD 22;
      L     LD 18;
      T     W [AR1,P#100.0];
END_FUNCTION

FUNCTION "DosLine" : VOID	// FC 91
VERSION : 0.1
BEGIN
// (block stored without names or comments; labels and parameter names are numbered)
NETWORK
TITLE =
      L     #PARAM1;
      BLD   5;
      T     LD 3;
      TAK;
      T     LD 7;
      L     P##PARAM12;
      LAR1;
      L     W [AR1,P#0.0];
      T     LW 1;
      OPN   DB [LW 1];
      L     D [AR1,P#2.0];
      LAR1;
      L     LD 7;
      L     LD 3;
      T     D [AR1,P#0.0];
      L     #PARAM2;
      BLD   5;
      T     LD 3;
      TAK;
      T     LD 7;
      L     P##PARAM12;
      LAR1;
      L     W [AR1,P#0.0];
      T     LW 1;
      OPN   DB [LW 1];
      L     D [AR1,P#2.0];
      LAR1;
      L     LD 7;
      L     LD 3;
      T     D [AR1,P#8.0];
      L     #PARAM3;
      BLD   5;
      T     LD 3;
      TAK;
      T     LD 7;
      L     P##PARAM12;
      LAR1;
      L     W [AR1,P#0.0];
      T     LW 1;
      OPN   DB [LW 1];
      L     D [AR1,P#2.0];
      LAR1;
      L     LD 7;
      L     LD 3;
      T     D [AR1,P#22.0];
      L     #PARAM4;
      BLD   5;
      T     LD 3;
      TAK;
      T     LD 7;
      L     P##PARAM12;
      LAR1;
      L     W [AR1,P#0.0];
      T     LW 1;
      OPN   DB [LW 1];
      L     D [AR1,P#2.0];
      LAR1;
      L     LD 7;
      L     LD 3;
      T     W [AR1,P#20.0];
      A     #PARAM6;
      BLD   5;
      T     LD 3;
      TAK;
      T     LD 7;
      L     P##PARAM12;
      LAR1;
      L     W [AR1,P#0.0];
      T     LW 1;
      OPN   DB [LW 1];
      L     D [AR1,P#2.0];
      LAR1;
      L     LD 7;
      L     LD 3;
      =      [AR1,P#32.4];
      L     #PARAM5;
      BLD   5;
      T     LD 3;
      TAK;
      T     LD 7;
      L     P##PARAM12;
      LAR1;
      L     W [AR1,P#0.0];
      T     LW 1;
      OPN   DB [LW 1];
      L     D [AR1,P#2.0];
      LAR1;
      L     LD 7;
      L     LD 3;
      T     W [AR1,P#30.0];
      BLD   5;
      T     LD 3;
      TAK;
      T     LD 7;
      L     P##PARAM12;
      LAR1;
      L     W [AR1,P#0.0];
      T     LW 1;
      OPN   DB [LW 1];
      L     D [AR1,P#2.0];
      LAR1;
      L     LD 7;
      L     LD 3;
      L     D [AR1,P#4.0];
      T     #PARAM7;
      BLD   5;
      T     LD 3;
      TAK;
      T     LD 7;
      L     P##PARAM12;
      LAR1;
      L     W [AR1,P#0.0];
      T     LW 1;
      OPN   DB [LW 1];
      L     D [AR1,P#2.0];
      LAR1;
      L     LD 7;
      L     LD 3;
      A      [AR1,P#32.3];
      =     #PARAM9;
      BLD   5;
      T     LD 3;
      TAK;
      T     LD 7;
      L     P##PARAM12;
      LAR1;
      L     W [AR1,P#0.0];
      T     LW 1;
      OPN   DB [LW 1];
      L     D [AR1,P#2.0];
      LAR1;
      L     LD 7;
      L     LD 3;
      L     D [AR1,P#26.0];
      T     #PARAM8;
      BLD   5;
      T     LD 3;
      TAK;
      T     LD 7;
      L     P##PARAM12;
      LAR1;
      L     W [AR1,P#0.0];
      T     LW 1;
      OPN   DB [LW 1];
      L     D [AR1,P#2.0];
      LAR1;
      L     LD 7;
      L     LD 3;
      A      [AR1,P#32.0];
      =     #PARAM10;
      BLD   5;
      T     LD 3;
      TAK;
      T     LD 7;
      L     P##PARAM12;
      LAR1;
      L     W [AR1,P#0.0];
      T     LW 1;
      OPN   DB [LW 1];
      L     D [AR1,P#2.0];
      LAR1;
      L     LD 7;
      L     LD 3;
      A      [AR1,P#32.1];
      =     #PARAM11;
END_FUNCTION

FUNCTION "AUTO_VALVE" : VOID	// FC 100
AUTHOR : gaw-be
FAMILY : VALVE
NAME : VALVE_A
VERSION : 0.1
BEGIN
// (block stored without names or comments; labels and parameter names are numbered)
NETWORK
TITLE =
      BLD   5;
      T     LD 103;
      TAK;
      T     LD 107;
      L     P##PARAM10;
      LAR1;
      L     W [AR1,P#0.0];
      T     LW 101;
      OPN   DB [LW 101];
      L     D [AR1,P#2.0];
      LAR1;
      L     LD 107;
      L     LD 103;
      L     W [AR1,P#2.0];
      L     -1;
      ==I;
      BLD   5;
      T     LD 103;
      TAK;
      T     LD 107;
      L     P##PARAM10;
      LAR1;
      L     W [AR1,P#0.0];
      T     LW 101;
      OPN   DB [LW 101];
      L     D [AR1,P#2.0];
      LAR1;
      L     LD 107;
      L     LD 103;
      R      [AR1,P#4.0];
      L     #PARAM6;
      BLD   5;
      T     LD 103;
      TAK;
      T     LD 107;
      L     P##PARAM10;
      LAR1;
      L     W [AR1,P#0.0];
      T     LW 101;
      OPN   DB [LW 101];
      L     D [AR1,P#2.0];
      LAR1;
      L     LD 107;
      L     LD 103;
      L     W [AR1,P#2.0];
      <>I;
      JC    M002;
      BLD   5;
      T     LD 103;
      TAK;
      T     LD 107;
      L     P##PARAM10;
      LAR1;
      L     W [AR1,P#0.0];
      T     LW 101;
      OPN   DB [LW 101];
      L     D [AR1,P#2.0];
      LAR1;
      L     LD 107;
      L     LD 103;
      A      [AR1,P#4.0];
      JC    M001;
      BLD   5;
      T     LD 103;
      TAK;
      T     LD 107;
      L     P##PARAM9;
      LAR1;
      L     W [AR1,P#0.0];
      T     LW 101;
      OPN   DB [LW 101];
      L     D [AR1,P#2.0];
      LAR1;
      L     LD 107;
      L     LD 103;
      A      [AR1,P#0.0];
      BLD   5;
      T     LD 103;
      TAK;
      T     LD 107;
      L     P##PARAM10;
      LAR1;
      L     W [AR1,P#0.0];
      T     LW 101;
      OPN   DB [LW 101];
      L     D [AR1,P#2.0];
      LAR1;
      L     LD 107;
      L     LD 103;
      =      [AR1,P#0.0];
      BLD   5;
      T     LD 103;
      TAK;
      T     LD 107;
      L     P##PARAM9;
      LAR1;
      L     W [AR1,P#0.0];
      T     LW 101;
      OPN   DB [LW 101];
      L     D [AR1,P#2.0];
      LAR1;
      L     LD 107;
      L     LD 103;
      A      [AR1,P#0.1];
      BLD   5;
      T     LD 103;
      TAK;
      T     LD 107;
      L     P##PARAM10;
      LAR1;
      L     W [AR1,P#0.0];
      T     LW 101;
      OPN   DB [LW 101];
      L     D [AR1,P#2.0];
      LAR1;
      L     LD 107;
      L     LD 103;
      =      [AR1,P#0.1];
      SET;
      BLD   5;
      T     LD 103;
      TAK;
      T     LD 107;
      L     P##PARAM10;
      LAR1;
      L     W [AR1,P#0.0];
      T     LW 101;
      OPN   DB [LW 101];
      L     D [AR1,P#2.0];
      LAR1;
      L     LD 107;
      L     LD 103;
      =      [AR1,P#4.0];
M001: BLD   5;
      T     LD 103;
      TAK;
      T     LD 107;
      L     P##PARAM10;
      LAR1;
      L     W [AR1,P#0.0];
      T     LW 101;
      OPN   DB [LW 101];
      L     D [AR1,P#2.0];
      LAR1;
      L     LD 107;
      L     LD 103;
      A      [AR1,P#0.0];
      BLD   5;
      T     LD 103;
      TAK;
      T     LD 107;
      L     P##PARAM9;
      LAR1;
      L     W [AR1,P#0.0];
      T     LW 101;
      OPN   DB [LW 101];
      L     D [AR1,P#2.0];
      LAR1;
      L     LD 107;
      L     LD 103;
      =      [AR1,P#0.0];
      BLD   5;
      T     LD 103;
      TAK;
      T     LD 107;
      L     P##PARAM10;
      LAR1;
      L     W [AR1,P#0.0];
      T     LW 101;
      OPN   DB [LW 101];
      L     D [AR1,P#2.0];
      LAR1;
      L     LD 107;
      L     LD 103;
      A      [AR1,P#0.1];
      BLD   5;
      T     LD 103;
      TAK;
      T     LD 107;
      L     P##PARAM9;
      LAR1;
      L     W [AR1,P#0.0];
      T     LW 101;
      OPN   DB [LW 101];
      L     D [AR1,P#2.0];
      LAR1;
      L     LD 107;
      L     LD 103;
      =      [AR1,P#0.1];
      BLD   5;
      T     LD 103;
      TAK;
      T     LD 107;
      L     P##PARAM9;
      LAR1;
      L     W [AR1,P#0.0];
      T     LW 101;
      OPN   DB [LW 101];
      L     D [AR1,P#2.0];
      LAR1;
      L     LD 107;
      L     LD 103;
      A      [AR1,P#0.2];
      BLD   5;
      T     LD 103;
      TAK;
      T     LD 107;
      L     P##PARAM10;
      LAR1;
      L     W [AR1,P#0.0];
      T     LW 101;
      OPN   DB [LW 101];
      L     D [AR1,P#2.0];
      LAR1;
      L     LD 107;
      L     LD 103;
      =      [AR1,P#0.2];
      BLD   5;
      T     LD 103;
      TAK;
      T     LD 107;
      L     P##PARAM9;
      LAR1;
      L     W [AR1,P#0.0];
      T     LW 101;
      OPN   DB [LW 101];
      L     D [AR1,P#2.0];
      LAR1;
      L     LD 107;
      L     LD 103;
      A      [AR1,P#0.3];
      BLD   5;
      T     LD 103;
      TAK;
      T     LD 107;
      L     P##PARAM10;
      LAR1;
      L     W [AR1,P#0.0];
      T     LW 101;
      OPN   DB [LW 101];
      L     D [AR1,P#2.0];
      LAR1;
      L     LD 107;
      L     LD 103;
      =      [AR1,P#0.3];
      BLD   5;
      T     LD 103;
      TAK;
      T     LD 107;
      L     P##PARAM9;
      LAR1;
      L     W [AR1,P#0.0];
      T     LW 101;
      OPN   DB [LW 101];
      L     D [AR1,P#2.0];
      LAR1;
      L     LD 107;
      L     LD 103;
      A      [AR1,P#0.4];
      BLD   5;
      T     LD 103;
      TAK;
      T     LD 107;
      L     P##PARAM10;
      LAR1;
      L     W [AR1,P#0.0];
      T     LW 101;
      OPN   DB [LW 101];
      L     D [AR1,P#2.0];
      LAR1;
      L     LD 107;
      L     LD 103;
      =      [AR1,P#0.4];
      BLD   5;
      T     LD 103;
      TAK;
      T     LD 107;
      L     P##PARAM9;
      LAR1;
      L     W [AR1,P#0.0];
      T     LW 101;
      OPN   DB [LW 101];
      L     D [AR1,P#2.0];
      LAR1;
      L     LD 107;
      L     LD 103;
      A      [AR1,P#0.5];
      BLD   5;
      T     LD 103;
      TAK;
      T     LD 107;
      L     P##PARAM10;
      LAR1;
      L     W [AR1,P#0.0];
      T     LW 101;
      OPN   DB [LW 101];
      L     D [AR1,P#2.0];
      LAR1;
      L     LD 107;
      L     LD 103;
      =      [AR1,P#0.5];
      BLD   5;
      T     LD 103;
      TAK;
      T     LD 107;
      L     P##PARAM9;
      LAR1;
      L     W [AR1,P#0.0];
      T     LW 101;
      OPN   DB [LW 101];
      L     D [AR1,P#2.0];
      LAR1;
      L     LD 107;
      L     LD 103;
      A      [AR1,P#0.6];
      BLD   5;
      T     LD 103;
      TAK;
      T     LD 107;
      L     P##PARAM10;
      LAR1;
      L     W [AR1,P#0.0];
      T     LW 101;
      OPN   DB [LW 101];
      L     D [AR1,P#2.0];
      LAR1;
      L     LD 107;
      L     LD 103;
      =      [AR1,P#0.6];
      BLD   5;
      T     LD 103;
      TAK;
      T     LD 107;
      L     P##PARAM9;
      LAR1;
      L     W [AR1,P#0.0];
      T     LW 101;
      OPN   DB [LW 101];
      L     D [AR1,P#2.0];
      LAR1;
      L     LD 107;
      L     LD 103;
      A      [AR1,P#0.7];
      BLD   5;
      T     LD 103;
      TAK;
      T     LD 107;
      L     P##PARAM10;
      LAR1;
      L     W [AR1,P#0.0];
      T     LW 101;
      OPN   DB [LW 101];
      L     D [AR1,P#2.0];
      LAR1;
      L     LD 107;
      L     LD 103;
      =      [AR1,P#0.7];
      BLD   5;
      T     LD 103;
      TAK;
      T     LD 107;
      L     P##PARAM9;
      LAR1;
      L     W [AR1,P#0.0];
      T     LW 101;
      OPN   DB [LW 101];
      L     D [AR1,P#2.0];
      LAR1;
      L     LD 107;
      L     LD 103;
      L     B [AR1,P#1.0];
      BLD   5;
      T     LD 103;
      TAK;
      T     LD 107;
      L     P##PARAM10;
      LAR1;
      L     W [AR1,P#0.0];
      T     LW 101;
      OPN   DB [LW 101];
      L     D [AR1,P#2.0];
      LAR1;
      L     LD 107;
      L     LD 103;
      T     B [AR1,P#1.0];
M002: NOP   0;
NETWORK
TITLE =
      A     #PARAM1;
      BLD   5;
      T     LD 103;
      TAK;
      T     LD 107;
      L     P##PARAM9;
      LAR1;
      L     W [AR1,P#0.0];
      T     LW 101;
      OPN   DB [LW 101];
      L     D [AR1,P#2.0];
      LAR1;
      L     LD 107;
      L     LD 103;
      =      [AR1,P#0.2];
NETWORK
TITLE =
      A     #PARAM2;
      BLD   5;
      T     LD 103;
      TAK;
      T     LD 107;
      L     P##PARAM9;
      LAR1;
      L     W [AR1,P#0.0];
      T     LW 101;
      OPN   DB [LW 101];
      L     D [AR1,P#2.0];
      LAR1;
      L     LD 107;
      L     LD 103;
      =      [AR1,P#0.3];
NETWORK
TITLE =
      A(;
      A     #PARAM4;
      BLD   5;
      T     LD 103;
      TAK;
      T     LD 107;
      L     P##PARAM9;
      LAR1;
      L     W [AR1,P#0.0];
      T     LW 101;
      OPN   DB [LW 101];
      L     D [AR1,P#2.0];
      LAR1;
      L     LD 107;
      L     LD 103;
      AN     [AR1,P#0.0];
      O;
      BLD   5;
      T     LD 103;
      TAK;
      T     LD 107;
      L     P##PARAM9;
      LAR1;
      L     W [AR1,P#0.0];
      T     LW 101;
      OPN   DB [LW 101];
      L     D [AR1,P#2.0];
      LAR1;
      L     LD 107;
      L     LD 103;
      A      [AR1,P#0.0];
      BLD   5;
      T     LD 103;
      TAK;
      T     LD 107;
      L     P##PARAM9;
      LAR1;
      L     W [AR1,P#0.0];
      T     LW 101;
      OPN   DB [LW 101];
      L     D [AR1,P#2.0];
      LAR1;
      L     LD 107;
      L     LD 103;
      A      [AR1,P#0.1];
      );
      AN    #PARAM5;
      =     #PARAM7;
      =     L 0.0;
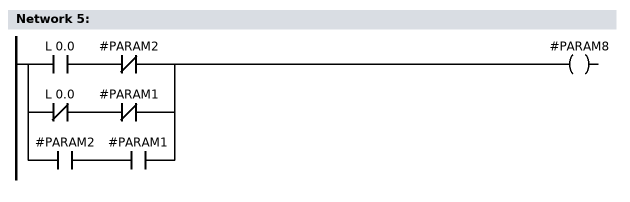
NETWORK
TITLE =
      A     L 0.0;
      AN    #PARAM2;
      O;
      AN    L 0.0;
      AN    #PARAM1;
      O;
      A     #PARAM2;
      A     #PARAM1;
      =     #PARAM8;
NETWORK
TITLE =
      A(;
      A     #PARAM1;
      AN    L 0.0;
      O;
      AN    #PARAM1;
      AN    L 0.0;
      AN    M 0.7;
      );
      A(;
      A     #PARAM2;
      A     #PARAM1;
      NOT;
      );
      BLD   5;
      T     LD 103;
      TAK;
      T     LD 107;
      L     P##PARAM9;
      LAR1;
      L     W [AR1,P#0.0];
      T     LW 101;
      OPN   DB [LW 101];
      L     D [AR1,P#2.0];
      LAR1;
      L     LD 107;
      L     LD 103;
      =      [AR1,P#0.4];
NETWORK
TITLE =
      A(;
      A     #PARAM2;
      A     L 0.0;
      O;
      AN    #PARAM2;
      A     L 0.0;
      AN    M 0.7;
      );
      A(;
      A     #PARAM2;
      A     #PARAM1;
      NOT;
      );
      BLD   5;
      T     LD 103;
      TAK;
      T     LD 107;
      L     P##PARAM9;
      LAR1;
      L     W [AR1,P#0.0];
      T     LW 101;
      OPN   DB [LW 101];
      L     D [AR1,P#2.0];
      LAR1;
      L     LD 107;
      L     LD 103;
      =      [AR1,P#0.5];
NETWORK
TITLE =
      A(;
      AN    #PARAM1;
      AN    L 0.0;
      O;
      AN    #PARAM2;
      A     L 0.0;
      );
      A     #PARAM3;
      A     M 0.7;
      O;
      A     #PARAM2;
      A     #PARAM1;
      A     M 0.7;
      BLD   5;
      T     LD 103;
      TAK;
      T     LD 107;
      L     P##PARAM9;
      LAR1;
      L     W [AR1,P#0.0];
      T     LW 101;
      OPN   DB [LW 101];
      L     D [AR1,P#2.0];
      LAR1;
      L     LD 107;
      L     LD 103;
      =      [AR1,P#0.6];
NETWORK
TITLE =
      A(;
      AN    #PARAM1;
      AN    L 0.0;
      O;
      AN    #PARAM2;
      A     L 0.0;
      );
      AN    #PARAM3;
      A     M 0.7;
      O;
      A     #PARAM2;
      A     #PARAM1;
      AN    M 0.7;
      BLD   5;
      T     LD 103;
      TAK;
      T     LD 107;
      L     P##PARAM9;
      LAR1;
      L     W [AR1,P#0.0];
      T     LW 101;
      OPN   DB [LW 101];
      L     D [AR1,P#2.0];
      LAR1;
      L     LD 107;
      L     LD 103;
      =      [AR1,P#0.7];
NETWORK
TITLE =
      BLD   5;
      T     LD 103;
      TAK;
      T     LD 107;
      L     P##PARAM9;
      LAR1;
      L     W [AR1,P#0.0];
      T     LW 101;
      OPN   DB [LW 101];
      L     D [AR1,P#2.0];
      LAR1;
      L     LD 107;
      L     LD 103;
      A      [AR1,P#0.0];
      =     L 100.0;
      BLD   5;
      T     LD 103;
      TAK;
      T     LD 107;
      L     P##PARAM9;
      LAR1;
      L     W [AR1,P#0.0];
      T     LW 101;
      OPN   DB [LW 101];
      L     D [AR1,P#2.0];
      LAR1;
      L     LD 107;
      L     LD 103;
      A      [AR1,P#0.1];
      =     L 100.1;
      BLD   5;
      T     LD 103;
      TAK;
      T     LD 107;
      L     P##PARAM9;
      LAR1;
      L     W [AR1,P#0.0];
      T     LW 101;
      OPN   DB [LW 101];
      L     D [AR1,P#2.0];
      LAR1;
      L     LD 107;
      L     LD 103;
      A      [AR1,P#0.2];
      =     L 100.2;
      BLD   5;
      T     LD 103;
      TAK;
      T     LD 107;
      L     P##PARAM9;
      LAR1;
      L     W [AR1,P#0.0];
      T     LW 101;
      OPN   DB [LW 101];
      L     D [AR1,P#2.0];
      LAR1;
      L     LD 107;
      L     LD 103;
      A      [AR1,P#0.3];
      =     L 100.3;
      BLD   5;
      T     LD 103;
      TAK;
      T     LD 107;
      L     P##PARAM9;
      LAR1;
      L     W [AR1,P#0.0];
      T     LW 101;
      OPN   DB [LW 101];
      L     D [AR1,P#2.0];
      LAR1;
      L     LD 107;
      L     LD 103;
      A      [AR1,P#0.4];
      =     L 100.4;
      BLD   5;
      T     LD 103;
      TAK;
      T     LD 107;
      L     P##PARAM9;
      LAR1;
      L     W [AR1,P#0.0];
      T     LW 101;
      OPN   DB [LW 101];
      L     D [AR1,P#2.0];
      LAR1;
      L     LD 107;
      L     LD 103;
      A      [AR1,P#0.5];
      =     L 100.5;
      BLD   5;
      T     LD 103;
      TAK;
      T     LD 107;
      L     P##PARAM9;
      LAR1;
      L     W [AR1,P#0.0];
      T     LW 101;
      OPN   DB [LW 101];
      L     D [AR1,P#2.0];
      LAR1;
      L     LD 107;
      L     LD 103;
      A      [AR1,P#0.6];
      =     L 100.6;
      BLD   5;
      T     LD 103;
      TAK;
      T     LD 107;
      L     P##PARAM9;
      LAR1;
      L     W [AR1,P#0.0];
      T     LW 101;
      OPN   DB [LW 101];
      L     D [AR1,P#2.0];
      LAR1;
      L     LD 107;
      L     LD 103;
      A      [AR1,P#0.7];
      =     L 100.7;
      L     LB 100;
      BLD   5;
      T     LD 103;
      TAK;
      T     LD 107;
      L     P##PARAM9;
      LAR1;
      L     W [AR1,P#0.0];
      T     LW 101;
      OPN   DB [LW 101];
      L     D [AR1,P#2.0];
      LAR1;
      L     LD 107;
      L     LD 103;
      T     B [AR1,P#1.0];
END_FUNCTION

